CONFIGURATION Config0
  VAR_GLOBAL
    F_Conf : BOOL := TRUE;  (* Флаг конфигурирования *)
    F_Res : BOOL := FALSE;  (* Флаг готовности результата *)
    STAT : TStat;  (* Состояние выполнения *)
    HDR : THead;  (* Заголовок модели *)
    STS : TSets;  (* Массивы настроек *)
    ITS : TItems;  (* Массивы элементов *)
    SFC : ARRAY[0..2] OF TItem := [0, 0, 0];  (* Массив поверхностей *)
    CFG : TConf;  (* Заголовок трансформатора *)
    RAD : ARRAY[0..15] OF TRad := [0, 0, 0, 0, 0, 0, 0, 0, 0, 0, 0, 0, 0, 0, 0, 0];  (* Массив радиаторов *)
    VRI : TVarI;  (* Заголовок входа (24 байт) *)
    PHI : ARRAY[0..2] OF TPhaseI := [0, 0, 0];  (* Вход по фазам (3x32 байт) *)
    VRO : TVarO;  (* Заголовок выхода (24 байт) *)
    PHO : ARRAY[0..2] OF TPhaseO := [0, 0, 0];  (* Выход по фазам (3x32 байт) *)
    RES : TRes;  (* Заголовок расчёта *)
    rTest : REAL := 0.0;  (* Для отладки *)
  END_VAR
  RESOURCE Res0 ON PLC
    VAR_GLOBAL RETAIN
      MW0 AT %MW0 : UINT := 16#0000;  (* DEF[0].ID: = Трансформатор = *)
      MW1 AT %MW1 : UINT := 16#8000;  (* DEF[0].CF: Флаги (СК|ось|форма) *)
      MW2 AT %MW2 : UINT := 0;  (* DEF[0].R0: Начальный радиус *)
      MW3 AT %MW3 : UINT := 0;  (* DEF[0].XYZ[0]: Координата X *)
      MW4 AT %MW4 : UINT := 0;  (* DEF[0].XYZ[1]: Координата Y *)
      MW5 AT %MW5 : UINT := 0;  (* DEF[0].XYZ[2]: Координата Z *)
      MW6 AT %MW6 : UINT := 3600;  (* DEF[0].LWH[0]: Длина L *)
      MW7 AT %MW7 : UINT := 1240;  (* DEF[0].LWH[1]: Ширина W *)
      MW8 AT %MW8 : UINT := 3150;  (* DEF[0].LWH[2]: Высота H *)
      MW9 AT %MW9 : UINT := 16#7000;  (* DEF[0].GMV: #Grd(4)|#Mat(4)|#Val(8) *)
      MW10 AT %MW10 : UINT := 16#1000;  (* DEF[1].ID: = КОЖУХ = *)
      MW11 AT %MW11 : UINT := 16#8000;  (* DEF[1].CF: Флаги (СК|ось|форма) *)
      MW12 AT %MW12 : UINT := 0;  (* DEF[1].R0: Начальный радиус *)
      MW13 AT %MW13 : UINT := 0;  (* DEF[1].XYZ[0]: Координата X *)
      MW14 AT %MW14 : UINT := 0;  (* DEF[1].XYZ[1]: Координата Y *)
      MW15 AT %MW15 : UINT := 0;  (* DEF[1].XYZ[2]: Координата Z *)
      MW16 AT %MW16 : UINT := 3600;  (* DEF[1].LWH[0]: Длина L *)
      MW17 AT %MW17 : UINT := 1240;  (* DEF[1].LWH[1]: Ширина W *)
      MW18 AT %MW18 : UINT := 3150;  (* DEF[1].LWH[2]: Высота H *)
      MW19 AT %MW19 : UINT := 16#8000;  (* DEF[1].GMV: #Grd(4)|#Mat(4)|#Val(8) *)
      MW20 AT %MW20 : UINT := 16#1100;  (* DEF[2].ID: - Крышка (центр) *)
      MW21 AT %MW21 : UINT := 16#0000;  (* DEF[2].CF: Флаги (СК|ось|форма) *)
      MW22 AT %MW22 : UINT := 0;  (* DEF[2].R0: Начальный радиус *)
      MW23 AT %MW23 : UINT := 620;  (* DEF[2].XYZ[0]: Координата X *)
      MW24 AT %MW24 : UINT := 0;  (* DEF[2].XYZ[1]: Координата Y *)
      MW25 AT %MW25 : UINT := 3140;  (* DEF[2].XYZ[2]: Координата Z *)
      MW26 AT %MW26 : UINT := 2360;  (* DEF[2].LWH[0]: Длина L *)
      MW27 AT %MW27 : UINT := 1240;  (* DEF[2].LWH[1]: Ширина W *)
      MW28 AT %MW28 : UINT := 10;  (* DEF[2].LWH[2]: Высота H *)
      MW29 AT %MW29 : UINT := 16#8200;  (* DEF[2].GMV: #Grd(4)|#Mat(4)|#Val(8) *)
      MW30 AT %MW30 : UINT := 16#1200;  (* DEF[3].ID: - Крышка (лев) *)
      MW31 AT %MW31 : UINT := 16#7400;  (* DEF[3].CF: Флаги (СК|ось|форма) *)
      MW32 AT %MW32 : UINT := 0;  (* DEF[3].R0: Начальный радиус *)
      MW33 AT %MW33 : UINT := 620;  (* DEF[3].XYZ[0]: Координата X *)
      MW34 AT %MW34 : UINT := 620;  (* DEF[3].XYZ[1]: Координата Y *)
      MW35 AT %MW35 : UINT := 3140;  (* DEF[3].XYZ[2]: Координата Z *)
      MW36 AT %MW36 : UINT := 620;  (* DEF[3].LWH[0]: Длина L *)
      MW37 AT %MW37 : UINT := 180;  (* DEF[3].LWH[1]: Ширина W *)
      MW38 AT %MW38 : UINT := 10;  (* DEF[3].LWH[2]: Высота H *)
      MW39 AT %MW39 : UINT := 16#3200;  (* DEF[3].GMV: #Grd(4)|#Mat(4)|#Val(8) *)
      MW40 AT %MW40 : UINT := 16#1300;  (* DEF[4].ID: - Крышка (прав) *)
      MW41 AT %MW41 : UINT := 16#7C00;  (* DEF[4].CF: Флаги (СК|ось|форма) *)
      MW42 AT %MW42 : UINT := 0;  (* DEF[4].R0: Начальный радиус *)
      MW43 AT %MW43 : UINT := 2980;  (* DEF[4].XYZ[0]: Координата X *)
      MW44 AT %MW44 : UINT := 620;  (* DEF[4].XYZ[1]: Координата Y *)
      MW45 AT %MW45 : UINT := 3140;  (* DEF[4].XYZ[2]: Координата Z *)
      MW46 AT %MW46 : UINT := 620;  (* DEF[4].LWH[0]: Длина L *)
      MW47 AT %MW47 : UINT := 180;  (* DEF[4].LWH[1]: Ширина W *)
      MW48 AT %MW48 : UINT := 10;  (* DEF[4].LWH[2]: Высота H *)
      MW49 AT %MW49 : UINT := 16#3200;  (* DEF[4].GMV: #Grd(4)|#Mat(4)|#Val(8) *)
      MW50 AT %MW50 : UINT := 16#1400;  (* DEF[5].ID: - Днище (центр) *)
      MW51 AT %MW51 : UINT := 16#0000;  (* DEF[5].CF: Флаги (СК|ось|форма) *)
      MW52 AT %MW52 : UINT := 0;  (* DEF[5].R0: Начальный радиус *)
      MW53 AT %MW53 : UINT := 620;  (* DEF[5].XYZ[0]: Координата X *)
      MW54 AT %MW54 : UINT := 0;  (* DEF[5].XYZ[1]: Координата Y *)
      MW55 AT %MW55 : UINT := 0;  (* DEF[5].XYZ[2]: Координата Z *)
      MW56 AT %MW56 : UINT := 2360;  (* DEF[5].LWH[0]: Длина L *)
      MW57 AT %MW57 : UINT := 1240;  (* DEF[5].LWH[1]: Ширина W *)
      MW58 AT %MW58 : UINT := 10;  (* DEF[5].LWH[2]: Высота H *)
      MW59 AT %MW59 : UINT := 16#8200;  (* DEF[5].GMV: #Grd(4)|#Mat(4)|#Val(8) *)
      MW60 AT %MW60 : UINT := 16#1500;  (* DEF[6].ID: - Днище (лев) *)
      MW61 AT %MW61 : UINT := 16#7400;  (* DEF[6].CF: Флаги (СК|ось|форма) *)
      MW62 AT %MW62 : UINT := 0;  (* DEF[6].R0: Начальный радиус *)
      MW63 AT %MW63 : UINT := 620;  (* DEF[6].XYZ[0]: Координата X *)
      MW64 AT %MW64 : UINT := 620;  (* DEF[6].XYZ[1]: Координата Y *)
      MW65 AT %MW65 : UINT := 0;  (* DEF[6].XYZ[2]: Координата Z *)
      MW66 AT %MW66 : UINT := 620;  (* DEF[6].LWH[0]: Длина L *)
      MW67 AT %MW67 : UINT := 180;  (* DEF[6].LWH[1]: Ширина W *)
      MW68 AT %MW68 : UINT := 10;  (* DEF[6].LWH[2]: Высота H *)
      MW69 AT %MW69 : UINT := 16#3200;  (* DEF[6].GMV: #Grd(4)|#Mat(4)|#Val(8) *)
      MW70 AT %MW70 : UINT := 16#1600;  (* DEF[7].ID: - Днище (прав) *)
      MW71 AT %MW71 : UINT := 16#7C00;  (* DEF[7].CF: Флаги (СК|ось|форма) *)
      MW72 AT %MW72 : UINT := 0;  (* DEF[7].R0: Начальный радиус *)
      MW73 AT %MW73 : UINT := 2980;  (* DEF[7].XYZ[0]: Координата X *)
      MW74 AT %MW74 : UINT := 620;  (* DEF[7].XYZ[1]: Координата Y *)
      MW75 AT %MW75 : UINT := 0;  (* DEF[7].XYZ[2]: Координата Z *)
      MW76 AT %MW76 : UINT := 620;  (* DEF[7].LWH[0]: Длина L *)
      MW77 AT %MW77 : UINT := 180;  (* DEF[7].LWH[1]: Ширина W *)
      MW78 AT %MW78 : UINT := 10;  (* DEF[7].LWH[2]: Высота H *)
      MW79 AT %MW79 : UINT := 16#3200;  (* DEF[7].GMV: #Grd(4)|#Mat(4)|#Val(8) *)
      MW80 AT %MW80 : UINT := 16#1700;  (* DEF[8].ID: - Стенка левая *)
      MW81 AT %MW81 : UINT := 16#7400;  (* DEF[8].CF: Флаги (СК|ось|форма) *)
      MW82 AT %MW82 : UINT := 610;  (* DEF[8].R0: Начальный радиус *)
      MW83 AT %MW83 : UINT := 620;  (* DEF[8].XYZ[0]: Координата X *)
      MW84 AT %MW84 : UINT := 620;  (* DEF[8].XYZ[1]: Координата Y *)
      MW85 AT %MW85 : UINT := 10;  (* DEF[8].XYZ[2]: Координата Z *)
      MW86 AT %MW86 : UINT := 10;  (* DEF[8].LWH[0]: Длина L *)
      MW87 AT %MW87 : UINT := 180;  (* DEF[8].LWH[1]: Ширина W *)
      MW88 AT %MW88 : UINT := 3130;  (* DEF[8].LWH[2]: Высота H *)
      MW89 AT %MW89 : UINT := 16#1200;  (* DEF[8].GMV: #Grd(4)|#Mat(4)|#Val(8) *)
      MW90 AT %MW90 : UINT := 16#1800;  (* DEF[9].ID: - Стенка правая *)
      MW91 AT %MW91 : UINT := 16#7C00;  (* DEF[9].CF: Флаги (СК|ось|форма) *)
      MW92 AT %MW92 : UINT := 610;  (* DEF[9].R0: Начальный радиус *)
      MW93 AT %MW93 : UINT := 2980;  (* DEF[9].XYZ[0]: Координата X *)
      MW94 AT %MW94 : UINT := 620;  (* DEF[9].XYZ[1]: Координата Y *)
      MW95 AT %MW95 : UINT := 10;  (* DEF[9].XYZ[2]: Координата Z *)
      MW96 AT %MW96 : UINT := 10;  (* DEF[9].LWH[0]: Длина L *)
      MW97 AT %MW97 : UINT := 180;  (* DEF[9].LWH[1]: Ширина W *)
      MW98 AT %MW98 : UINT := 3130;  (* DEF[9].LWH[2]: Высота H *)
      MW99 AT %MW99 : UINT := 16#1200;  (* DEF[9].GMV: #Grd(4)|#Mat(4)|#Val(8) *)
      MW100 AT %MW100 : UINT := 16#1900;  (* DEF[10].ID: - Стенка передняя *)
      MW101 AT %MW101 : UINT := 16#0000;  (* DEF[10].CF: Флаги (СК|ось|форма) *)
      MW102 AT %MW102 : UINT := 0;  (* DEF[10].R0: Начальный радиус *)
      MW103 AT %MW103 : UINT := 620;  (* DEF[10].XYZ[0]: Координата X *)
      MW104 AT %MW104 : UINT := 0;  (* DEF[10].XYZ[1]: Координата Y *)
      MW105 AT %MW105 : UINT := 10;  (* DEF[10].XYZ[2]: Координата Z *)
      MW106 AT %MW106 : UINT := 2360;  (* DEF[10].LWH[0]: Длина L *)
      MW107 AT %MW107 : UINT := 10;  (* DEF[10].LWH[1]: Ширина W *)
      MW108 AT %MW108 : UINT := 3130;  (* DEF[10].LWH[2]: Высота H *)
      MW109 AT %MW109 : UINT := 16#7200;  (* DEF[10].GMV: #Grd(4)|#Mat(4)|#Val(8) *)
      MW110 AT %MW110 : UINT := 16#1A00;  (* DEF[11].ID: - Стенка задняя *)
      MW111 AT %MW111 : UINT := 16#0000;  (* DEF[11].CF: Флаги (СК|ось|форма) *)
      MW112 AT %MW112 : UINT := 0;  (* DEF[11].R0: Начальный радиус *)
      MW113 AT %MW113 : UINT := 620;  (* DEF[11].XYZ[0]: Координата X *)
      MW114 AT %MW114 : UINT := 1230;  (* DEF[11].XYZ[1]: Координата Y *)
      MW115 AT %MW115 : UINT := 10;  (* DEF[11].XYZ[2]: Координата Z *)
      MW116 AT %MW116 : UINT := 2360;  (* DEF[11].LWH[0]: Длина L *)
      MW117 AT %MW117 : UINT := 10;  (* DEF[11].LWH[1]: Ширина W *)
      MW118 AT %MW118 : UINT := 3130;  (* DEF[11].LWH[2]: Высота H *)
      MW119 AT %MW119 : UINT := 16#7200;  (* DEF[11].GMV: #Grd(4)|#Mat(4)|#Val(8) *)
      MW120 AT %MW120 : UINT := 16#1B00;  (* DEF[12].ID: - Масло слева *)
      MW121 AT %MW121 : UINT := 16#7400;  (* DEF[12].CF: Флаги (СК|ось|форма) *)
      MW122 AT %MW122 : UINT := 590;  (* DEF[12].R0: Начальный радиус *)
      MW123 AT %MW123 : UINT := 620;  (* DEF[12].XYZ[0]: Координата X *)
      MW124 AT %MW124 : UINT := 620;  (* DEF[12].XYZ[1]: Координата Y *)
      MW125 AT %MW125 : UINT := 10;  (* DEF[12].XYZ[2]: Координата Z *)
      MW126 AT %MW126 : UINT := 20;  (* DEF[12].LWH[0]: Длина L *)
      MW127 AT %MW127 : UINT := 180;  (* DEF[12].LWH[1]: Ширина W *)
      MW128 AT %MW128 : UINT := 3130;  (* DEF[12].LWH[2]: Высота H *)
      MW129 AT %MW129 : UINT := 16#1100;  (* DEF[12].GMV: #Grd(4)|#Mat(4)|#Val(8) *)
      MW130 AT %MW130 : UINT := 16#1C00;  (* DEF[13].ID: - Масло справа *)
      MW131 AT %MW131 : UINT := 16#7C00;  (* DEF[13].CF: Флаги (СК|ось|форма) *)
      MW132 AT %MW132 : UINT := 590;  (* DEF[13].R0: Начальный радиус *)
      MW133 AT %MW133 : UINT := 2980;  (* DEF[13].XYZ[0]: Координата X *)
      MW134 AT %MW134 : UINT := 620;  (* DEF[13].XYZ[1]: Координата Y *)
      MW135 AT %MW135 : UINT := 10;  (* DEF[13].XYZ[2]: Координата Z *)
      MW136 AT %MW136 : UINT := 20;  (* DEF[13].LWH[0]: Длина L *)
      MW137 AT %MW137 : UINT := 180;  (* DEF[13].LWH[1]: Ширина W *)
      MW138 AT %MW138 : UINT := 3130;  (* DEF[13].LWH[2]: Высота H *)
      MW139 AT %MW139 : UINT := 16#1100;  (* DEF[13].GMV: #Grd(4)|#Mat(4)|#Val(8) *)
      MW140 AT %MW140 : UINT := 16#1D00;  (* DEF[14].ID: - Масло спереди *)
      MW141 AT %MW141 : UINT := 16#0000;  (* DEF[14].CF: Флаги (СК|ось|форма) *)
      MW142 AT %MW142 : UINT := 0;  (* DEF[14].R0: Начальный радиус *)
      MW143 AT %MW143 : UINT := 620;  (* DEF[14].XYZ[0]: Координата X *)
      MW144 AT %MW144 : UINT := 10;  (* DEF[14].XYZ[1]: Координата Y *)
      MW145 AT %MW145 : UINT := 10;  (* DEF[14].XYZ[2]: Координата Z *)
      MW146 AT %MW146 : UINT := 2360;  (* DEF[14].LWH[0]: Длина L *)
      MW147 AT %MW147 : UINT := 20;  (* DEF[14].LWH[1]: Ширина W *)
      MW148 AT %MW148 : UINT := 3130;  (* DEF[14].LWH[2]: Высота H *)
      MW149 AT %MW149 : UINT := 16#7100;  (* DEF[14].GMV: #Grd(4)|#Mat(4)|#Val(8) *)
      MW150 AT %MW150 : UINT := 16#1E00;  (* DEF[15].ID: - Масло сзади *)
      MW151 AT %MW151 : UINT := 16#0000;  (* DEF[15].CF: Флаги (СК|ось|форма) *)
      MW152 AT %MW152 : UINT := 0;  (* DEF[15].R0: Начальный радиус *)
      MW153 AT %MW153 : UINT := 620;  (* DEF[15].XYZ[0]: Координата X *)
      MW154 AT %MW154 : UINT := 1210;  (* DEF[15].XYZ[1]: Координата Y *)
      MW155 AT %MW155 : UINT := 10;  (* DEF[15].XYZ[2]: Координата Z *)
      MW156 AT %MW156 : UINT := 2360;  (* DEF[15].LWH[0]: Длина L *)
      MW157 AT %MW157 : UINT := 20;  (* DEF[15].LWH[1]: Ширина W *)
      MW158 AT %MW158 : UINT := 3130;  (* DEF[15].LWH[2]: Высота H *)
      MW159 AT %MW159 : UINT := 16#7100;  (* DEF[15].GMV: #Grd(4)|#Mat(4)|#Val(8) *)
      MW160 AT %MW160 : UINT := 16#2000;  (* DEF[16].ID: = ЧЕРДАК = *)
      MW161 AT %MW161 : UINT := 16#8000;  (* DEF[16].CF: Флаги (СК|ось|форма) *)
      MW162 AT %MW162 : UINT := 0;  (* DEF[16].R0: Начальный радиус *)
      MW163 AT %MW163 : UINT := 30;  (* DEF[16].XYZ[0]: Координата X *)
      MW164 AT %MW164 : UINT := 30;  (* DEF[16].XYZ[1]: Координата Y *)
      MW165 AT %MW165 : UINT := 2400;  (* DEF[16].XYZ[2]: Координата Z *)
      MW166 AT %MW166 : UINT := 3540;  (* DEF[16].LWH[0]: Длина L *)
      MW167 AT %MW167 : UINT := 1180;  (* DEF[16].LWH[1]: Ширина W *)
      MW168 AT %MW168 : UINT := 740;  (* DEF[16].LWH[2]: Высота H *)
      MW169 AT %MW169 : UINT := 16#8000;  (* DEF[16].GMV: #Grd(4)|#Mat(4)|#Val(8) *)
      MW170 AT %MW170 : UINT := 16#2100;  (* DEF[17].ID: - Масло верх (центр) *)
      MW171 AT %MW171 : UINT := 16#0000;  (* DEF[17].CF: Флаги (СК|ось|форма) *)
      MW172 AT %MW172 : UINT := 0;  (* DEF[17].R0: Начальный радиус *)
      MW173 AT %MW173 : UINT := 590;  (* DEF[17].XYZ[0]: Координата X *)
      MW174 AT %MW174 : UINT := 0;  (* DEF[17].XYZ[1]: Координата Y *)
      MW175 AT %MW175 : UINT := 350;  (* DEF[17].XYZ[2]: Координата Z *)
      MW176 AT %MW176 : UINT := 2360;  (* DEF[17].LWH[0]: Длина L *)
      MW177 AT %MW177 : UINT := 1180;  (* DEF[17].LWH[1]: Ширина W *)
      MW178 AT %MW178 : UINT := 390;  (* DEF[17].LWH[2]: Высота H *)
      MW179 AT %MW179 : UINT := 16#8100;  (* DEF[17].GMV: #Grd(4)|#Mat(4)|#Val(8) *)
      MW180 AT %MW180 : UINT := 16#2200;  (* DEF[18].ID: - Масло верх (лев) *)
      MW181 AT %MW181 : UINT := 16#7400;  (* DEF[18].CF: Флаги (СК|ось|форма) *)
      MW182 AT %MW182 : UINT := 0;  (* DEF[18].R0: Начальный радиус *)
      MW183 AT %MW183 : UINT := 590;  (* DEF[18].XYZ[0]: Координата X *)
      MW184 AT %MW184 : UINT := 590;  (* DEF[18].XYZ[1]: Координата Y *)
      MW185 AT %MW185 : UINT := 350;  (* DEF[18].XYZ[2]: Координата Z *)
      MW186 AT %MW186 : UINT := 590;  (* DEF[18].LWH[0]: Длина L *)
      MW187 AT %MW187 : UINT := 180;  (* DEF[18].LWH[1]: Ширина W *)
      MW188 AT %MW188 : UINT := 390;  (* DEF[18].LWH[2]: Высота H *)
      MW189 AT %MW189 : UINT := 16#3100;  (* DEF[18].GMV: #Grd(4)|#Mat(4)|#Val(8) *)
      MW190 AT %MW190 : UINT := 16#2300;  (* DEF[19].ID: - Масло верх (прав) *)
      MW191 AT %MW191 : UINT := 16#7C00;  (* DEF[19].CF: Флаги (СК|ось|форма) *)
      MW192 AT %MW192 : UINT := 0;  (* DEF[19].R0: Начальный радиус *)
      MW193 AT %MW193 : UINT := 2950;  (* DEF[19].XYZ[0]: Координата X *)
      MW194 AT %MW194 : UINT := 590;  (* DEF[19].XYZ[1]: Координата Y *)
      MW195 AT %MW195 : UINT := 350;  (* DEF[19].XYZ[2]: Координата Z *)
      MW196 AT %MW196 : UINT := 590;  (* DEF[19].LWH[0]: Длина L *)
      MW197 AT %MW197 : UINT := 180;  (* DEF[19].LWH[1]: Ширина W *)
      MW198 AT %MW198 : UINT := 390;  (* DEF[19].LWH[2]: Высота H *)
      MW199 AT %MW199 : UINT := 16#3100;  (* DEF[19].GMV: #Grd(4)|#Mat(4)|#Val(8) *)
      MW200 AT %MW200 : UINT := 16#2400;  (* DEF[20].ID: = Ярмовой слой (верх) = *)
      MW201 AT %MW201 : UINT := 16#8000;  (* DEF[20].CF: Флаги (СК|ось|форма) *)
      MW202 AT %MW202 : UINT := 0;  (* DEF[20].R0: Начальный радиус *)
      MW203 AT %MW203 : UINT := 0;  (* DEF[20].XYZ[0]: Координата X *)
      MW204 AT %MW204 : UINT := 0;  (* DEF[20].XYZ[1]: Координата Y *)
      MW205 AT %MW205 : UINT := 0;  (* DEF[20].XYZ[2]: Координата Z *)
      MW206 AT %MW206 : UINT := 3540;  (* DEF[20].LWH[0]: Длина L *)
      MW207 AT %MW207 : UINT := 1180;  (* DEF[20].LWH[1]: Ширина W *)
      MW208 AT %MW208 : UINT := 350;  (* DEF[20].LWH[2]: Высота H *)
      MW209 AT %MW209 : UINT := 16#8000;  (* DEF[20].GMV: #Grd(4)|#Mat(4)|#Val(8) *)
      MW210 AT %MW210 : UINT := 16#2410;  (* DEF[21].ID: - Ярмо (верх) *)
      MW211 AT %MW211 : UINT := 16#0000;  (* DEF[21].CF: Флаги (СК|ось|форма) *)
      MW212 AT %MW212 : UINT := 0;  (* DEF[21].R0: Начальный радиус *)
      MW213 AT %MW213 : UINT := 275;  (* DEF[21].XYZ[0]: Координата X *)
      MW214 AT %MW214 : UINT := 275;  (* DEF[21].XYZ[1]: Координата Y *)
      MW215 AT %MW215 : UINT := 0;  (* DEF[21].XYZ[2]: Координата Z *)
      MW216 AT %MW216 : UINT := 2990;  (* DEF[21].LWH[0]: Длина L *)
      MW217 AT %MW217 : UINT := 630;  (* DEF[21].LWH[1]: Ширина W *)
      MW218 AT %MW218 : UINT := 350;  (* DEF[21].LWH[2]: Высота H *)
      MW219 AT %MW219 : UINT := 16#8300;  (* DEF[21].GMV: #Grd(4)|#Mat(4)|#Val(8) *)
      MW220 AT %MW220 : UINT := 16#2420;  (* DEF[22].ID: - Масло слева (верх) *)
      MW221 AT %MW221 : UINT := 16#7460;  (* DEF[22].CF: Флаги (СК|ось|форма) *)
      MW222 AT %MW222 : UINT := 315;  (* DEF[22].R0: Начальный радиус *)
      MW223 AT %MW223 : UINT := 590;  (* DEF[22].XYZ[0]: Координата X *)
      MW224 AT %MW224 : UINT := 590;  (* DEF[22].XYZ[1]: Координата Y *)
      MW225 AT %MW225 : UINT := 0;  (* DEF[22].XYZ[2]: Координата Z *)
      MW226 AT %MW226 : UINT := 275;  (* DEF[22].LWH[0]: Длина L *)
      MW227 AT %MW227 : UINT := 180;  (* DEF[22].LWH[1]: Ширина W *)
      MW228 AT %MW228 : UINT := 350;  (* DEF[22].LWH[2]: Высота H *)
      MW229 AT %MW229 : UINT := 16#3100;  (* DEF[22].GMV: #Grd(4)|#Mat(4)|#Val(8) *)
      MW230 AT %MW230 : UINT := 16#2430;  (* DEF[23].ID: - Масло справа (верх) *)
      MW231 AT %MW231 : UINT := 16#7C90;  (* DEF[23].CF: Флаги (СК|ось|форма) *)
      MW232 AT %MW232 : UINT := 315;  (* DEF[23].R0: Начальный радиус *)
      MW233 AT %MW233 : UINT := 2950;  (* DEF[23].XYZ[0]: Координата X *)
      MW234 AT %MW234 : UINT := 590;  (* DEF[23].XYZ[1]: Координата Y *)
      MW235 AT %MW235 : UINT := 0;  (* DEF[23].XYZ[2]: Координата Z *)
      MW236 AT %MW236 : UINT := 275;  (* DEF[23].LWH[0]: Длина L *)
      MW237 AT %MW237 : UINT := 180;  (* DEF[23].LWH[1]: Ширина W *)
      MW238 AT %MW238 : UINT := 350;  (* DEF[23].LWH[2]: Высота H *)
      MW239 AT %MW239 : UINT := 16#3100;  (* DEF[23].GMV: #Grd(4)|#Mat(4)|#Val(8) *)
      MW240 AT %MW240 : UINT := 16#2440;  (* DEF[24].ID: - Масло спереди (верх) *)
      MW241 AT %MW241 : UINT := 16#0000;  (* DEF[24].CF: Флаги (СК|ось|форма) *)
      MW242 AT %MW242 : UINT := 0;  (* DEF[24].R0: Начальный радиус *)
      MW243 AT %MW243 : UINT := 590;  (* DEF[24].XYZ[0]: Координата X *)
      MW244 AT %MW244 : UINT := 0;  (* DEF[24].XYZ[1]: Координата Y *)
      MW245 AT %MW245 : UINT := 0;  (* DEF[24].XYZ[2]: Координата Z *)
      MW246 AT %MW246 : UINT := 2360;  (* DEF[24].LWH[0]: Длина L *)
      MW247 AT %MW247 : UINT := 275;  (* DEF[24].LWH[1]: Ширина W *)
      MW248 AT %MW248 : UINT := 350;  (* DEF[24].LWH[2]: Высота H *)
      MW249 AT %MW249 : UINT := 16#8100;  (* DEF[24].GMV: #Grd(4)|#Mat(4)|#Val(8) *)
      MW250 AT %MW250 : UINT := 16#2450;  (* DEF[25].ID: - Масло сзади (верх) *)
      MW251 AT %MW251 : UINT := 16#0000;  (* DEF[25].CF: Флаги (СК|ось|форма) *)
      MW252 AT %MW252 : UINT := 0;  (* DEF[25].R0: Начальный радиус *)
      MW253 AT %MW253 : UINT := 590;  (* DEF[25].XYZ[0]: Координата X *)
      MW254 AT %MW254 : UINT := 905;  (* DEF[25].XYZ[1]: Координата Y *)
      MW255 AT %MW255 : UINT := 0;  (* DEF[25].XYZ[2]: Координата Z *)
      MW256 AT %MW256 : UINT := 2360;  (* DEF[25].LWH[0]: Длина L *)
      MW257 AT %MW257 : UINT := 275;  (* DEF[25].LWH[1]: Ширина W *)
      MW258 AT %MW258 : UINT := 350;  (* DEF[25].LWH[2]: Высота H *)
      MW259 AT %MW259 : UINT := 16#8100;  (* DEF[25].GMV: #Grd(4)|#Mat(4)|#Val(8) *)
      MW260 AT %MW260 : UINT := 16#3000;  (* DEF[26].ID: = ЦОКОЛЬ = *)
      MW261 AT %MW261 : UINT := 16#8000;  (* DEF[26].CF: Флаги (СК|ось|форма) *)
      MW262 AT %MW262 : UINT := 0;  (* DEF[26].R0: Начальный радиус *)
      MW263 AT %MW263 : UINT := 30;  (* DEF[26].XYZ[0]: Координата X *)
      MW264 AT %MW264 : UINT := 30;  (* DEF[26].XYZ[1]: Координата Y *)
      MW265 AT %MW265 : UINT := 10;  (* DEF[26].XYZ[2]: Координата Z *)
      MW266 AT %MW266 : UINT := 3540;  (* DEF[26].LWH[0]: Длина L *)
      MW267 AT %MW267 : UINT := 1180;  (* DEF[26].LWH[1]: Ширина W *)
      MW268 AT %MW268 : UINT := 390;  (* DEF[26].LWH[2]: Высота H *)
      MW269 AT %MW269 : UINT := 16#8000;  (* DEF[26].GMV: #Grd(4)|#Mat(4)|#Val(8) *)
      MW270 AT %MW270 : UINT := 16#3100;  (* DEF[27].ID: - Масло низ (центр) *)
      MW271 AT %MW271 : UINT := 16#0000;  (* DEF[27].CF: Флаги (СК|ось|форма) *)
      MW272 AT %MW272 : UINT := 0;  (* DEF[27].R0: Начальный радиус *)
      MW273 AT %MW273 : UINT := 590;  (* DEF[27].XYZ[0]: Координата X *)
      MW274 AT %MW274 : UINT := 0;  (* DEF[27].XYZ[1]: Координата Y *)
      MW275 AT %MW275 : UINT := 0;  (* DEF[27].XYZ[2]: Координата Z *)
      MW276 AT %MW276 : UINT := 2360;  (* DEF[27].LWH[0]: Длина L *)
      MW277 AT %MW277 : UINT := 1180;  (* DEF[27].LWH[1]: Ширина W *)
      MW278 AT %MW278 : UINT := 40;  (* DEF[27].LWH[2]: Высота H *)
      MW279 AT %MW279 : UINT := 16#8100;  (* DEF[27].GMV: #Grd(4)|#Mat(4)|#Val(8) *)
      MW280 AT %MW280 : UINT := 16#3200;  (* DEF[28].ID: - Масло низ (лев) *)
      MW281 AT %MW281 : UINT := 16#7400;  (* DEF[28].CF: Флаги (СК|ось|форма) *)
      MW282 AT %MW282 : UINT := 0;  (* DEF[28].R0: Начальный радиус *)
      MW283 AT %MW283 : UINT := 590;  (* DEF[28].XYZ[0]: Координата X *)
      MW284 AT %MW284 : UINT := 590;  (* DEF[28].XYZ[1]: Координата Y *)
      MW285 AT %MW285 : UINT := 0;  (* DEF[28].XYZ[2]: Координата Z *)
      MW286 AT %MW286 : UINT := 590;  (* DEF[28].LWH[0]: Длина L *)
      MW287 AT %MW287 : UINT := 180;  (* DEF[28].LWH[1]: Ширина W *)
      MW288 AT %MW288 : UINT := 40;  (* DEF[28].LWH[2]: Высота H *)
      MW289 AT %MW289 : UINT := 16#3100;  (* DEF[28].GMV: #Grd(4)|#Mat(4)|#Val(8) *)
      MW290 AT %MW290 : UINT := 16#3300;  (* DEF[29].ID: - Масло низ (прав) *)
      MW291 AT %MW291 : UINT := 16#7C00;  (* DEF[29].CF: Флаги (СК|ось|форма) *)
      MW292 AT %MW292 : UINT := 0;  (* DEF[29].R0: Начальный радиус *)
      MW293 AT %MW293 : UINT := 2950;  (* DEF[29].XYZ[0]: Координата X *)
      MW294 AT %MW294 : UINT := 590;  (* DEF[29].XYZ[1]: Координата Y *)
      MW295 AT %MW295 : UINT := 0;  (* DEF[29].XYZ[2]: Координата Z *)
      MW296 AT %MW296 : UINT := 590;  (* DEF[29].LWH[0]: Длина L *)
      MW297 AT %MW297 : UINT := 180;  (* DEF[29].LWH[1]: Ширина W *)
      MW298 AT %MW298 : UINT := 40;  (* DEF[29].LWH[2]: Высота H *)
      MW299 AT %MW299 : UINT := 16#3100;  (* DEF[29].GMV: #Grd(4)|#Mat(4)|#Val(8) *)
      MW300 AT %MW300 : UINT := 16#3400;  (* DEF[30].ID: = Ярмовой слой (низ) = *)
      MW301 AT %MW301 : UINT := 16#8000;  (* DEF[30].CF: Флаги (СК|ось|форма) *)
      MW302 AT %MW302 : UINT := 0;  (* DEF[30].R0: Начальный радиус *)
      MW303 AT %MW303 : UINT := 0;  (* DEF[30].XYZ[0]: Координата X *)
      MW304 AT %MW304 : UINT := 0;  (* DEF[30].XYZ[1]: Координата Y *)
      MW305 AT %MW305 : UINT := 40;  (* DEF[30].XYZ[2]: Координата Z *)
      MW306 AT %MW306 : UINT := 3540;  (* DEF[30].LWH[0]: Длина L *)
      MW307 AT %MW307 : UINT := 1180;  (* DEF[30].LWH[1]: Ширина W *)
      MW308 AT %MW308 : UINT := 350;  (* DEF[30].LWH[2]: Высота H *)
      MW309 AT %MW309 : UINT := 16#8000;  (* DEF[30].GMV: #Grd(4)|#Mat(4)|#Val(8) *)
      MW310 AT %MW310 : UINT := 16#3410;  (* DEF[31].ID: - Ярмо (низ) *)
      MW311 AT %MW311 : UINT := 16#0000;  (* DEF[31].CF: Флаги (СК|ось|форма) *)
      MW312 AT %MW312 : UINT := 0;  (* DEF[31].R0: Начальный радиус *)
      MW313 AT %MW313 : UINT := 275;  (* DEF[31].XYZ[0]: Координата X *)
      MW314 AT %MW314 : UINT := 275;  (* DEF[31].XYZ[1]: Координата Y *)
      MW315 AT %MW315 : UINT := 0;  (* DEF[31].XYZ[2]: Координата Z *)
      MW316 AT %MW316 : UINT := 2990;  (* DEF[31].LWH[0]: Длина L *)
      MW317 AT %MW317 : UINT := 630;  (* DEF[31].LWH[1]: Ширина W *)
      MW318 AT %MW318 : UINT := 350;  (* DEF[31].LWH[2]: Высота H *)
      MW319 AT %MW319 : UINT := 16#8300;  (* DEF[31].GMV: #Grd(4)|#Mat(4)|#Val(8) *)
      MW320 AT %MW320 : UINT := 16#3420;  (* DEF[32].ID: - Масло слева (низ) *)
      MW321 AT %MW321 : UINT := 16#7460;  (* DEF[32].CF: Флаги (СК|ось|форма) *)
      MW322 AT %MW322 : UINT := 315;  (* DEF[32].R0: Начальный радиус *)
      MW323 AT %MW323 : UINT := 590;  (* DEF[32].XYZ[0]: Координата X *)
      MW324 AT %MW324 : UINT := 590;  (* DEF[32].XYZ[1]: Координата Y *)
      MW325 AT %MW325 : UINT := 0;  (* DEF[32].XYZ[2]: Координата Z *)
      MW326 AT %MW326 : UINT := 275;  (* DEF[32].LWH[0]: Длина L *)
      MW327 AT %MW327 : UINT := 180;  (* DEF[32].LWH[1]: Ширина W *)
      MW328 AT %MW328 : UINT := 350;  (* DEF[32].LWH[2]: Высота H *)
      MW329 AT %MW329 : UINT := 16#3100;  (* DEF[32].GMV: #Grd(4)|#Mat(4)|#Val(8) *)
      MW330 AT %MW330 : UINT := 16#3430;  (* DEF[33].ID: - Масло справа (низ) *)
      MW331 AT %MW331 : UINT := 16#7C90;  (* DEF[33].CF: Флаги (СК|ось|форма) *)
      MW332 AT %MW332 : UINT := 315;  (* DEF[33].R0: Начальный радиус *)
      MW333 AT %MW333 : UINT := 2950;  (* DEF[33].XYZ[0]: Координата X *)
      MW334 AT %MW334 : UINT := 590;  (* DEF[33].XYZ[1]: Координата Y *)
      MW335 AT %MW335 : UINT := 0;  (* DEF[33].XYZ[2]: Координата Z *)
      MW336 AT %MW336 : UINT := 275;  (* DEF[33].LWH[0]: Длина L *)
      MW337 AT %MW337 : UINT := 180;  (* DEF[33].LWH[1]: Ширина W *)
      MW338 AT %MW338 : UINT := 350;  (* DEF[33].LWH[2]: Высота H *)
      MW339 AT %MW339 : UINT := 16#3100;  (* DEF[33].GMV: #Grd(4)|#Mat(4)|#Val(8) *)
      MW340 AT %MW340 : UINT := 16#3440;  (* DEF[34].ID: - Масло спереди (низ) *)
      MW341 AT %MW341 : UINT := 16#0000;  (* DEF[34].CF: Флаги (СК|ось|форма) *)
      MW342 AT %MW342 : UINT := 0;  (* DEF[34].R0: Начальный радиус *)
      MW343 AT %MW343 : UINT := 590;  (* DEF[34].XYZ[0]: Координата X *)
      MW344 AT %MW344 : UINT := 0;  (* DEF[34].XYZ[1]: Координата Y *)
      MW345 AT %MW345 : UINT := 0;  (* DEF[34].XYZ[2]: Координата Z *)
      MW346 AT %MW346 : UINT := 2360;  (* DEF[34].LWH[0]: Длина L *)
      MW347 AT %MW347 : UINT := 275;  (* DEF[34].LWH[1]: Ширина W *)
      MW348 AT %MW348 : UINT := 350;  (* DEF[34].LWH[2]: Высота H *)
      MW349 AT %MW349 : UINT := 16#8100;  (* DEF[34].GMV: #Grd(4)|#Mat(4)|#Val(8) *)
      MW350 AT %MW350 : UINT := 16#3450;  (* DEF[35].ID: - Масло сзади (низ) *)
      MW351 AT %MW351 : UINT := 16#0000;  (* DEF[35].CF: Флаги (СК|ось|форма) *)
      MW352 AT %MW352 : UINT := 0;  (* DEF[35].R0: Начальный радиус *)
      MW353 AT %MW353 : UINT := 590;  (* DEF[35].XYZ[0]: Координата X *)
      MW354 AT %MW354 : UINT := 905;  (* DEF[35].XYZ[1]: Координата Y *)
      MW355 AT %MW355 : UINT := 0;  (* DEF[35].XYZ[2]: Координата Z *)
      MW356 AT %MW356 : UINT := 2360;  (* DEF[35].LWH[0]: Длина L *)
      MW357 AT %MW357 : UINT := 275;  (* DEF[35].LWH[1]: Ширина W *)
      MW358 AT %MW358 : UINT := 350;  (* DEF[35].LWH[2]: Высота H *)
      MW359 AT %MW359 : UINT := 16#8100;  (* DEF[35].GMV: #Grd(4)|#Mat(4)|#Val(8) *)
      MW360 AT %MW360 : UINT := 16#4000;  (* DEF[36].ID: = АКТИВНАЯ ЗОНА = *)
      MW361 AT %MW361 : UINT := 16#8000;  (* DEF[36].CF: Флаги (СК|ось|форма) *)
      MW362 AT %MW362 : UINT := 0;  (* DEF[36].R0: Начальный радиус *)
      MW363 AT %MW363 : UINT := 30;  (* DEF[36].XYZ[0]: Координата X *)
      MW364 AT %MW364 : UINT := 30;  (* DEF[36].XYZ[1]: Координата Y *)
      MW365 AT %MW365 : UINT := 400;  (* DEF[36].XYZ[2]: Координата Z *)
      MW366 AT %MW366 : UINT := 3540;  (* DEF[36].LWH[0]: Длина L *)
      MW367 AT %MW367 : UINT := 1180;  (* DEF[36].LWH[1]: Ширина W *)
      MW368 AT %MW368 : UINT := 2000;  (* DEF[36].LWH[2]: Высота H *)
      MW369 AT %MW369 : UINT := 16#8000;  (* DEF[36].GMV: #Grd(4)|#Mat(4)|#Val(8) *)
      MW370 AT %MW370 : UINT := 16#4100;  (* DEF[37].ID: = Фаза 1 (лев) = *)
      MW371 AT %MW371 : UINT := 16#F009;  (* DEF[37].CF: Флаги (СК|ось|форма) *)
      MW372 AT %MW372 : UINT := 0;  (* DEF[37].R0: Начальный радиус *)
      MW373 AT %MW373 : UINT := 590;  (* DEF[37].XYZ[0]: Координата X *)
      MW374 AT %MW374 : UINT := 590;  (* DEF[37].XYZ[1]: Координата Y *)
      MW375 AT %MW375 : UINT := 0;  (* DEF[37].XYZ[2]: Координата Z *)
      MW376 AT %MW376 : UINT := 590;  (* DEF[37].LWH[0]: Длина L *)
      MW377 AT %MW377 : UINT := 360;  (* DEF[37].LWH[1]: Ширина W *)
      MW378 AT %MW378 : UINT := 2000;  (* DEF[37].LWH[2]: Высота H *)
      MW379 AT %MW379 : UINT := 16#1000;  (* DEF[37].GMV: #Grd(4)|#Mat(4)|#Val(8) *)
      MW380 AT %MW380 : UINT := 16#4110;  (* DEF[38].ID: - Стержень *)
      MW381 AT %MW381 : UINT := 16#4000;  (* DEF[38].CF: Флаги (СК|ось|форма) *)
      MW382 AT %MW382 : UINT := 0;  (* DEF[38].R0: Начальный радиус *)
      MW383 AT %MW383 : UINT := 0;  (* DEF[38].XYZ[0]: Координата X *)
      MW384 AT %MW384 : UINT := 0;  (* DEF[38].XYZ[1]: Координата Y *)
      MW385 AT %MW385 : UINT := 0;  (* DEF[38].XYZ[2]: Координата Z *)
      MW386 AT %MW386 : UINT := 315;  (* DEF[38].LWH[0]: Длина L *)
      MW387 AT %MW387 : UINT := 360;  (* DEF[38].LWH[1]: Ширина W *)
      MW388 AT %MW388 : UINT := 2000;  (* DEF[38].LWH[2]: Высота H *)
      MW389 AT %MW389 : UINT := 16#1300;  (* DEF[38].GMV: #Grd(4)|#Mat(4)|#Val(8) *)
      MW390 AT %MW390 : UINT := 16#4120;  (* DEF[39].ID: - Масло сверху *)
      MW391 AT %MW391 : UINT := 16#4009;  (* DEF[39].CF: Флаги (СК|ось|форма) *)
      MW392 AT %MW392 : UINT := 0;  (* DEF[39].R0: Начальный радиус *)
      MW393 AT %MW393 : UINT := 315;  (* DEF[39].XYZ[0]: Координата X *)
      MW394 AT %MW394 : UINT := 0;  (* DEF[39].XYZ[1]: Координата Y *)
      MW395 AT %MW395 : UINT := 1850;  (* DEF[39].XYZ[2]: Координата Z *)
      MW396 AT %MW396 : UINT := 275;  (* DEF[39].LWH[0]: Длина L *)
      MW397 AT %MW397 : UINT := 360;  (* DEF[39].LWH[1]: Ширина W *)
      MW398 AT %MW398 : UINT := 150;  (* DEF[39].LWH[2]: Высота H *)
      MW399 AT %MW399 : UINT := 16#5100;  (* DEF[39].GMV: #Grd(4)|#Mat(4)|#Val(8) *)
      MW400 AT %MW400 : UINT := 16#4130;  (* DEF[40].ID: - Масло снизу *)
      MW401 AT %MW401 : UINT := 16#4009;  (* DEF[40].CF: Флаги (СК|ось|форма) *)
      MW402 AT %MW402 : UINT := 0;  (* DEF[40].R0: Начальный радиус *)
      MW403 AT %MW403 : UINT := 315;  (* DEF[40].XYZ[0]: Координата X *)
      MW404 AT %MW404 : UINT := 0;  (* DEF[40].XYZ[1]: Координата Y *)
      MW405 AT %MW405 : UINT := 0;  (* DEF[40].XYZ[2]: Координата Z *)
      MW406 AT %MW406 : UINT := 275;  (* DEF[40].LWH[0]: Длина L *)
      MW407 AT %MW407 : UINT := 360;  (* DEF[40].LWH[1]: Ширина W *)
      MW408 AT %MW408 : UINT := 150;  (* DEF[40].LWH[2]: Высота H *)
      MW409 AT %MW409 : UINT := 16#5100;  (* DEF[40].GMV: #Grd(4)|#Mat(4)|#Val(8) *)
      MW410 AT %MW410 : UINT := 16#4140;  (* DEF[41].ID: - Маслоканал-1 *)
      MW411 AT %MW411 : UINT := 16#4000;  (* DEF[41].CF: Флаги (СК|ось|форма) *)
      MW412 AT %MW412 : UINT := 0;  (* DEF[41].R0: Начальный радиус *)
      MW413 AT %MW413 : UINT := 315;  (* DEF[41].XYZ[0]: Координата X *)
      MW414 AT %MW414 : UINT := 0;  (* DEF[41].XYZ[1]: Координата Y *)
      MW415 AT %MW415 : UINT := 150;  (* DEF[41].XYZ[2]: Координата Z *)
      MW416 AT %MW416 : UINT := 30;  (* DEF[41].LWH[0]: Длина L *)
      MW417 AT %MW417 : UINT := 360;  (* DEF[41].LWH[1]: Ширина W *)
      MW418 AT %MW418 : UINT := 1700;  (* DEF[41].LWH[2]: Высота H *)
      MW419 AT %MW419 : UINT := 16#1100;  (* DEF[41].GMV: #Grd(4)|#Mat(4)|#Val(8) *)
      MW420 AT %MW420 : UINT := 16#4150;  (* DEF[42].ID: - Обмотка НН *)
      MW421 AT %MW421 : UINT := 16#4000;  (* DEF[42].CF: Флаги (СК|ось|форма) *)
      MW422 AT %MW422 : UINT := 0;  (* DEF[42].R0: Начальный радиус *)
      MW423 AT %MW423 : UINT := 345;  (* DEF[42].XYZ[0]: Координата X *)
      MW424 AT %MW424 : UINT := 0;  (* DEF[42].XYZ[1]: Координата Y *)
      MW425 AT %MW425 : UINT := 150;  (* DEF[42].XYZ[2]: Координата Z *)
      MW426 AT %MW426 : UINT := 80;  (* DEF[42].LWH[0]: Длина L *)
      MW427 AT %MW427 : UINT := 360;  (* DEF[42].LWH[1]: Ширина W *)
      MW428 AT %MW428 : UINT := 1700;  (* DEF[42].LWH[2]: Высота H *)
      MW429 AT %MW429 : UINT := 16#1400;  (* DEF[42].GMV: #Grd(4)|#Mat(4)|#Val(8) *)
      MW430 AT %MW430 : UINT := 16#4160;  (* DEF[43].ID: - Маслоканал-2 *)
      MW431 AT %MW431 : UINT := 16#4000;  (* DEF[43].CF: Флаги (СК|ось|форма) *)
      MW432 AT %MW432 : UINT := 0;  (* DEF[43].R0: Начальный радиус *)
      MW433 AT %MW433 : UINT := 425;  (* DEF[43].XYZ[0]: Координата X *)
      MW434 AT %MW434 : UINT := 0;  (* DEF[43].XYZ[1]: Координата Y *)
      MW435 AT %MW435 : UINT := 150;  (* DEF[43].XYZ[2]: Координата Z *)
      MW436 AT %MW436 : UINT := 30;  (* DEF[43].LWH[0]: Длина L *)
      MW437 AT %MW437 : UINT := 360;  (* DEF[43].LWH[1]: Ширина W *)
      MW438 AT %MW438 : UINT := 1700;  (* DEF[43].LWH[2]: Высота H *)
      MW439 AT %MW439 : UINT := 16#1100;  (* DEF[43].GMV: #Grd(4)|#Mat(4)|#Val(8) *)
      MW440 AT %MW440 : UINT := 16#4170;  (* DEF[44].ID: = Обмотка ВН = *)
      MW441 AT %MW441 : UINT := 16#C000;  (* DEF[44].CF: Флаги (СК|ось|форма) *)
      MW442 AT %MW442 : UINT := 0;  (* DEF[44].R0: Начальный радиус *)
      MW443 AT %MW443 : UINT := 455;  (* DEF[44].XYZ[0]: Координата X *)
      MW444 AT %MW444 : UINT := 0;  (* DEF[44].XYZ[1]: Координата Y *)
      MW445 AT %MW445 : UINT := 150;  (* DEF[44].XYZ[2]: Координата Z *)
      MW446 AT %MW446 : UINT := 90;  (* DEF[44].LWH[0]: Длина L *)
      MW447 AT %MW447 : UINT := 360;  (* DEF[44].LWH[1]: Ширина W *)
      MW448 AT %MW448 : UINT := 1700;  (* DEF[44].LWH[2]: Высота H *)
      MW449 AT %MW449 : UINT := 16#1000;  (* DEF[44].GMV: #Grd(4)|#Mat(4)|#Val(8) *)
      MW450 AT %MW450 : UINT := 16#4171;  (* DEF[45].ID: - Катушка ВН-1 *)
      MW451 AT %MW451 : UINT := 16#4000;  (* DEF[45].CF: Флаги (СК|ось|форма) *)
      MW452 AT %MW452 : UINT := 0;  (* DEF[45].R0: Начальный радиус *)
      MW453 AT %MW453 : UINT := 455;  (* DEF[45].XYZ[0]: Координата X *)
      MW454 AT %MW454 : UINT := 0;  (* DEF[45].XYZ[1]: Координата Y *)
      MW455 AT %MW455 : UINT := 150;  (* DEF[45].XYZ[2]: Координата Z *)
      MW456 AT %MW456 : UINT := 90;  (* DEF[45].LWH[0]: Длина L *)
      MW457 AT %MW457 : UINT := 360;  (* DEF[45].LWH[1]: Ширина W *)
      MW458 AT %MW458 : UINT := 170;  (* DEF[45].LWH[2]: Высота H *)
      MW459 AT %MW459 : UINT := 16#3500;  (* DEF[45].GMV: #Grd(4)|#Mat(4)|#Val(8) *)
      MW460 AT %MW460 : UINT := 16#4172;  (* DEF[46].ID: - Катушка ВН-2 *)
      MW461 AT %MW461 : UINT := 16#4000;  (* DEF[46].CF: Флаги (СК|ось|форма) *)
      MW462 AT %MW462 : UINT := 0;  (* DEF[46].R0: Начальный радиус *)
      MW463 AT %MW463 : UINT := 455;  (* DEF[46].XYZ[0]: Координата X *)
      MW464 AT %MW464 : UINT := 0;  (* DEF[46].XYZ[1]: Координата Y *)
      MW465 AT %MW465 : UINT := 320;  (* DEF[46].XYZ[2]: Координата Z *)
      MW466 AT %MW466 : UINT := 90;  (* DEF[46].LWH[0]: Длина L *)
      MW467 AT %MW467 : UINT := 360;  (* DEF[46].LWH[1]: Ширина W *)
      MW468 AT %MW468 : UINT := 170;  (* DEF[46].LWH[2]: Высота H *)
      MW469 AT %MW469 : UINT := 16#3500;  (* DEF[46].GMV: #Grd(4)|#Mat(4)|#Val(8) *)
      MW470 AT %MW470 : UINT := 16#4173;  (* DEF[47].ID: - Катушка ВН-3 *)
      MW471 AT %MW471 : UINT := 16#4000;  (* DEF[47].CF: Флаги (СК|ось|форма) *)
      MW472 AT %MW472 : UINT := 0;  (* DEF[47].R0: Начальный радиус *)
      MW473 AT %MW473 : UINT := 455;  (* DEF[47].XYZ[0]: Координата X *)
      MW474 AT %MW474 : UINT := 0;  (* DEF[47].XYZ[1]: Координата Y *)
      MW475 AT %MW475 : UINT := 490;  (* DEF[47].XYZ[2]: Координата Z *)
      MW476 AT %MW476 : UINT := 90;  (* DEF[47].LWH[0]: Длина L *)
      MW477 AT %MW477 : UINT := 360;  (* DEF[47].LWH[1]: Ширина W *)
      MW478 AT %MW478 : UINT := 170;  (* DEF[47].LWH[2]: Высота H *)
      MW479 AT %MW479 : UINT := 16#3500;  (* DEF[47].GMV: #Grd(4)|#Mat(4)|#Val(8) *)
      MW480 AT %MW480 : UINT := 16#4174;  (* DEF[48].ID: - Катушка ВН-4 *)
      MW481 AT %MW481 : UINT := 16#4000;  (* DEF[48].CF: Флаги (СК|ось|форма) *)
      MW482 AT %MW482 : UINT := 0;  (* DEF[48].R0: Начальный радиус *)
      MW483 AT %MW483 : UINT := 455;  (* DEF[48].XYZ[0]: Координата X *)
      MW484 AT %MW484 : UINT := 0;  (* DEF[48].XYZ[1]: Координата Y *)
      MW485 AT %MW485 : UINT := 660;  (* DEF[48].XYZ[2]: Координата Z *)
      MW486 AT %MW486 : UINT := 90;  (* DEF[48].LWH[0]: Длина L *)
      MW487 AT %MW487 : UINT := 360;  (* DEF[48].LWH[1]: Ширина W *)
      MW488 AT %MW488 : UINT := 170;  (* DEF[48].LWH[2]: Высота H *)
      MW489 AT %MW489 : UINT := 16#3500;  (* DEF[48].GMV: #Grd(4)|#Mat(4)|#Val(8) *)
      MW490 AT %MW490 : UINT := 16#4175;  (* DEF[49].ID: - Катушка ВН-5 *)
      MW491 AT %MW491 : UINT := 16#4000;  (* DEF[49].CF: Флаги (СК|ось|форма) *)
      MW492 AT %MW492 : UINT := 0;  (* DEF[49].R0: Начальный радиус *)
      MW493 AT %MW493 : UINT := 455;  (* DEF[49].XYZ[0]: Координата X *)
      MW494 AT %MW494 : UINT := 0;  (* DEF[49].XYZ[1]: Координата Y *)
      MW495 AT %MW495 : UINT := 830;  (* DEF[49].XYZ[2]: Координата Z *)
      MW496 AT %MW496 : UINT := 90;  (* DEF[49].LWH[0]: Длина L *)
      MW497 AT %MW497 : UINT := 360;  (* DEF[49].LWH[1]: Ширина W *)
      MW498 AT %MW498 : UINT := 170;  (* DEF[49].LWH[2]: Высота H *)
      MW499 AT %MW499 : UINT := 16#3500;  (* DEF[49].GMV: #Grd(4)|#Mat(4)|#Val(8) *)
      MW500 AT %MW500 : UINT := 16#4176;  (* DEF[50].ID: - Катушка ВН-6 *)
      MW501 AT %MW501 : UINT := 16#4000;  (* DEF[50].CF: Флаги (СК|ось|форма) *)
      MW502 AT %MW502 : UINT := 0;  (* DEF[50].R0: Начальный радиус *)
      MW503 AT %MW503 : UINT := 455;  (* DEF[50].XYZ[0]: Координата X *)
      MW504 AT %MW504 : UINT := 0;  (* DEF[50].XYZ[1]: Координата Y *)
      MW505 AT %MW505 : UINT := 1000;  (* DEF[50].XYZ[2]: Координата Z *)
      MW506 AT %MW506 : UINT := 90;  (* DEF[50].LWH[0]: Длина L *)
      MW507 AT %MW507 : UINT := 360;  (* DEF[50].LWH[1]: Ширина W *)
      MW508 AT %MW508 : UINT := 170;  (* DEF[50].LWH[2]: Высота H *)
      MW509 AT %MW509 : UINT := 16#3500;  (* DEF[50].GMV: #Grd(4)|#Mat(4)|#Val(8) *)
      MW510 AT %MW510 : UINT := 16#4177;  (* DEF[51].ID: - Катушка ВН-7 *)
      MW511 AT %MW511 : UINT := 16#4000;  (* DEF[51].CF: Флаги (СК|ось|форма) *)
      MW512 AT %MW512 : UINT := 0;  (* DEF[51].R0: Начальный радиус *)
      MW513 AT %MW513 : UINT := 455;  (* DEF[51].XYZ[0]: Координата X *)
      MW514 AT %MW514 : UINT := 0;  (* DEF[51].XYZ[1]: Координата Y *)
      MW515 AT %MW515 : UINT := 1170;  (* DEF[51].XYZ[2]: Координата Z *)
      MW516 AT %MW516 : UINT := 90;  (* DEF[51].LWH[0]: Длина L *)
      MW517 AT %MW517 : UINT := 360;  (* DEF[51].LWH[1]: Ширина W *)
      MW518 AT %MW518 : UINT := 170;  (* DEF[51].LWH[2]: Высота H *)
      MW519 AT %MW519 : UINT := 16#3500;  (* DEF[51].GMV: #Grd(4)|#Mat(4)|#Val(8) *)
      MW520 AT %MW520 : UINT := 16#4178;  (* DEF[52].ID: - Катушка ВН-8 *)
      MW521 AT %MW521 : UINT := 16#4000;  (* DEF[52].CF: Флаги (СК|ось|форма) *)
      MW522 AT %MW522 : UINT := 0;  (* DEF[52].R0: Начальный радиус *)
      MW523 AT %MW523 : UINT := 455;  (* DEF[52].XYZ[0]: Координата X *)
      MW524 AT %MW524 : UINT := 0;  (* DEF[52].XYZ[1]: Координата Y *)
      MW525 AT %MW525 : UINT := 1340;  (* DEF[52].XYZ[2]: Координата Z *)
      MW526 AT %MW526 : UINT := 90;  (* DEF[52].LWH[0]: Длина L *)
      MW527 AT %MW527 : UINT := 360;  (* DEF[52].LWH[1]: Ширина W *)
      MW528 AT %MW528 : UINT := 170;  (* DEF[52].LWH[2]: Высота H *)
      MW529 AT %MW529 : UINT := 16#3500;  (* DEF[52].GMV: #Grd(4)|#Mat(4)|#Val(8) *)
      MW530 AT %MW530 : UINT := 16#4179;  (* DEF[53].ID: - Катушка ВН-9 *)
      MW531 AT %MW531 : UINT := 16#4000;  (* DEF[53].CF: Флаги (СК|ось|форма) *)
      MW532 AT %MW532 : UINT := 0;  (* DEF[53].R0: Начальный радиус *)
      MW533 AT %MW533 : UINT := 455;  (* DEF[53].XYZ[0]: Координата X *)
      MW534 AT %MW534 : UINT := 0;  (* DEF[53].XYZ[1]: Координата Y *)
      MW535 AT %MW535 : UINT := 1510;  (* DEF[53].XYZ[2]: Координата Z *)
      MW536 AT %MW536 : UINT := 90;  (* DEF[53].LWH[0]: Длина L *)
      MW537 AT %MW537 : UINT := 360;  (* DEF[53].LWH[1]: Ширина W *)
      MW538 AT %MW538 : UINT := 170;  (* DEF[53].LWH[2]: Высота H *)
      MW539 AT %MW539 : UINT := 16#3500;  (* DEF[53].GMV: #Grd(4)|#Mat(4)|#Val(8) *)
      MW540 AT %MW540 : UINT := 16#417A;  (* DEF[54].ID: - Катушка ВН-10 *)
      MW541 AT %MW541 : UINT := 16#4000;  (* DEF[54].CF: Флаги (СК|ось|форма) *)
      MW542 AT %MW542 : UINT := 0;  (* DEF[54].R0: Начальный радиус *)
      MW543 AT %MW543 : UINT := 455;  (* DEF[54].XYZ[0]: Координата X *)
      MW544 AT %MW544 : UINT := 0;  (* DEF[54].XYZ[1]: Координата Y *)
      MW545 AT %MW545 : UINT := 1680;  (* DEF[54].XYZ[2]: Координата Z *)
      MW546 AT %MW546 : UINT := 90;  (* DEF[54].LWH[0]: Длина L *)
      MW547 AT %MW547 : UINT := 360;  (* DEF[54].LWH[1]: Ширина W *)
      MW548 AT %MW548 : UINT := 170;  (* DEF[54].LWH[2]: Высота H *)
      MW549 AT %MW549 : UINT := 16#3500;  (* DEF[54].GMV: #Grd(4)|#Mat(4)|#Val(8) *)
      MW550 AT %MW550 : UINT := 16#4180;  (* DEF[55].ID: = Маслоканал-3 = *)
      MW551 AT %MW551 : UINT := 16#C009;  (* DEF[55].CF: Флаги (СК|ось|форма) *)
      MW552 AT %MW552 : UINT := 0;  (* DEF[55].R0: Начальный радиус *)
      MW553 AT %MW553 : UINT := 545;  (* DEF[55].XYZ[0]: Координата X *)
      MW554 AT %MW554 : UINT := 0;  (* DEF[55].XYZ[1]: Координата Y *)
      MW555 AT %MW555 : UINT := 150;  (* DEF[55].XYZ[2]: Координата Z *)
      MW556 AT %MW556 : UINT := 45;  (* DEF[55].LWH[0]: Длина L *)
      MW557 AT %MW557 : UINT := 360;  (* DEF[55].LWH[1]: Ширина W *)
      MW558 AT %MW558 : UINT := 1700;  (* DEF[55].LWH[2]: Высота H *)
      MW559 AT %MW559 : UINT := 16#1000;  (* DEF[55].GMV: #Grd(4)|#Mat(4)|#Val(8) *)
      MW560 AT %MW560 : UINT := 16#4181;  (* DEF[56].ID: - Маслоканал-3 (лев) *)
      MW561 AT %MW561 : UINT := 16#4000;  (* DEF[56].CF: Флаги (СК|ось|форма) *)
      MW562 AT %MW562 : UINT := 0;  (* DEF[56].R0: Начальный радиус *)
      MW563 AT %MW563 : UINT := 545;  (* DEF[56].XYZ[0]: Координата X *)
      MW564 AT %MW564 : UINT := 90;  (* DEF[56].XYZ[1]: Координата Y *)
      MW565 AT %MW565 : UINT := 150;  (* DEF[56].XYZ[2]: Координата Z *)
      MW566 AT %MW566 : UINT := 45;  (* DEF[56].LWH[0]: Длина L *)
      MW567 AT %MW567 : UINT := 180;  (* DEF[56].LWH[1]: Ширина W *)
      MW568 AT %MW568 : UINT := 1700;  (* DEF[56].LWH[2]: Высота H *)
      MW569 AT %MW569 : UINT := 16#1100;  (* DEF[56].GMV: #Grd(4)|#Mat(4)|#Val(8) *)
      MW570 AT %MW570 : UINT := 16#4182;  (* DEF[57].ID: - Маслоканал-3 (прав) *)
      MW571 AT %MW571 : UINT := 16#4009;  (* DEF[57].CF: Флаги (СК|ось|форма) *)
      MW572 AT %MW572 : UINT := 0;  (* DEF[57].R0: Начальный радиус *)
      MW573 AT %MW573 : UINT := 545;  (* DEF[57].XYZ[0]: Координата X *)
      MW574 AT %MW574 : UINT := -90;  (* DEF[57].XYZ[1]: Координата Y *)
      MW575 AT %MW575 : UINT := 150;  (* DEF[57].XYZ[2]: Координата Z *)
      MW576 AT %MW576 : UINT := 45;  (* DEF[57].LWH[0]: Длина L *)
      MW577 AT %MW577 : UINT := 180;  (* DEF[57].LWH[1]: Ширина W *)
      MW578 AT %MW578 : UINT := 1700;  (* DEF[57].LWH[2]: Высота H *)
      MW579 AT %MW579 : UINT := 16#1100;  (* DEF[57].GMV: #Grd(4)|#Mat(4)|#Val(8) *)
      MW580 AT %MW580 : UINT := 16#4200;  (* DEF[58].ID: = Фаза 2 (центр) *)
      MW581 AT %MW581 : UINT := 16#F00F;  (* DEF[58].CF: Флаги (СК|ось|форма) *)
      MW582 AT %MW582 : UINT := 0;  (* DEF[58].R0: Начальный радиус *)
      MW583 AT %MW583 : UINT := 1770;  (* DEF[58].XYZ[0]: Координата X *)
      MW584 AT %MW584 : UINT := 590;  (* DEF[58].XYZ[1]: Координата Y *)
      MW585 AT %MW585 : UINT := 0;  (* DEF[58].XYZ[2]: Координата Z *)
      MW586 AT %MW586 : UINT := 590;  (* DEF[58].LWH[0]: Длина L *)
      MW587 AT %MW587 : UINT := 360;  (* DEF[58].LWH[1]: Ширина W *)
      MW588 AT %MW588 : UINT := 2000;  (* DEF[58].LWH[2]: Высота H *)
      MW589 AT %MW589 : UINT := 16#1000;  (* DEF[58].GMV: #Grd(4)|#Mat(4)|#Val(8) *)
      MW590 AT %MW590 : UINT := 16#4210;  (* DEF[59].ID: - Стержень *)
      MW591 AT %MW591 : UINT := 16#4000;  (* DEF[59].CF: Флаги (СК|ось|форма) *)
      MW592 AT %MW592 : UINT := 0;  (* DEF[59].R0: Начальный радиус *)
      MW593 AT %MW593 : UINT := 0;  (* DEF[59].XYZ[0]: Координата X *)
      MW594 AT %MW594 : UINT := 0;  (* DEF[59].XYZ[1]: Координата Y *)
      MW595 AT %MW595 : UINT := 0;  (* DEF[59].XYZ[2]: Координата Z *)
      MW596 AT %MW596 : UINT := 315;  (* DEF[59].LWH[0]: Длина L *)
      MW597 AT %MW597 : UINT := 360;  (* DEF[59].LWH[1]: Ширина W *)
      MW598 AT %MW598 : UINT := 2000;  (* DEF[59].LWH[2]: Высота H *)
      MW599 AT %MW599 : UINT := 16#1300;  (* DEF[59].GMV: #Grd(4)|#Mat(4)|#Val(8) *)
      MW600 AT %MW600 : UINT := 16#4220;  (* DEF[60].ID: - Масло сверху *)
      MW601 AT %MW601 : UINT := 16#400F;  (* DEF[60].CF: Флаги (СК|ось|форма) *)
      MW602 AT %MW602 : UINT := 0;  (* DEF[60].R0: Начальный радиус *)
      MW603 AT %MW603 : UINT := 315;  (* DEF[60].XYZ[0]: Координата X *)
      MW604 AT %MW604 : UINT := 0;  (* DEF[60].XYZ[1]: Координата Y *)
      MW605 AT %MW605 : UINT := 1850;  (* DEF[60].XYZ[2]: Координата Z *)
      MW606 AT %MW606 : UINT := 275;  (* DEF[60].LWH[0]: Длина L *)
      MW607 AT %MW607 : UINT := 360;  (* DEF[60].LWH[1]: Ширина W *)
      MW608 AT %MW608 : UINT := 150;  (* DEF[60].LWH[2]: Высота H *)
      MW609 AT %MW609 : UINT := 16#5100;  (* DEF[60].GMV: #Grd(4)|#Mat(4)|#Val(8) *)
      MW610 AT %MW610 : UINT := 16#4230;  (* DEF[61].ID: - Масло снизу *)
      MW611 AT %MW611 : UINT := 16#400F;  (* DEF[61].CF: Флаги (СК|ось|форма) *)
      MW612 AT %MW612 : UINT := 0;  (* DEF[61].R0: Начальный радиус *)
      MW613 AT %MW613 : UINT := 315;  (* DEF[61].XYZ[0]: Координата X *)
      MW614 AT %MW614 : UINT := 0;  (* DEF[61].XYZ[1]: Координата Y *)
      MW615 AT %MW615 : UINT := 0;  (* DEF[61].XYZ[2]: Координата Z *)
      MW616 AT %MW616 : UINT := 275;  (* DEF[61].LWH[0]: Длина L *)
      MW617 AT %MW617 : UINT := 360;  (* DEF[61].LWH[1]: Ширина W *)
      MW618 AT %MW618 : UINT := 150;  (* DEF[61].LWH[2]: Высота H *)
      MW619 AT %MW619 : UINT := 16#5100;  (* DEF[61].GMV: #Grd(4)|#Mat(4)|#Val(8) *)
      MW620 AT %MW620 : UINT := 16#4240;  (* DEF[62].ID: - Маслоканал-1 *)
      MW621 AT %MW621 : UINT := 16#4000;  (* DEF[62].CF: Флаги (СК|ось|форма) *)
      MW622 AT %MW622 : UINT := 0;  (* DEF[62].R0: Начальный радиус *)
      MW623 AT %MW623 : UINT := 315;  (* DEF[62].XYZ[0]: Координата X *)
      MW624 AT %MW624 : UINT := 0;  (* DEF[62].XYZ[1]: Координата Y *)
      MW625 AT %MW625 : UINT := 150;  (* DEF[62].XYZ[2]: Координата Z *)
      MW626 AT %MW626 : UINT := 30;  (* DEF[62].LWH[0]: Длина L *)
      MW627 AT %MW627 : UINT := 360;  (* DEF[62].LWH[1]: Ширина W *)
      MW628 AT %MW628 : UINT := 1700;  (* DEF[62].LWH[2]: Высота H *)
      MW629 AT %MW629 : UINT := 16#1100;  (* DEF[62].GMV: #Grd(4)|#Mat(4)|#Val(8) *)
      MW630 AT %MW630 : UINT := 16#4250;  (* DEF[63].ID: - Обмотка НН *)
      MW631 AT %MW631 : UINT := 16#4000;  (* DEF[63].CF: Флаги (СК|ось|форма) *)
      MW632 AT %MW632 : UINT := 0;  (* DEF[63].R0: Начальный радиус *)
      MW633 AT %MW633 : UINT := 345;  (* DEF[63].XYZ[0]: Координата X *)
      MW634 AT %MW634 : UINT := 0;  (* DEF[63].XYZ[1]: Координата Y *)
      MW635 AT %MW635 : UINT := 150;  (* DEF[63].XYZ[2]: Координата Z *)
      MW636 AT %MW636 : UINT := 80;  (* DEF[63].LWH[0]: Длина L *)
      MW637 AT %MW637 : UINT := 360;  (* DEF[63].LWH[1]: Ширина W *)
      MW638 AT %MW638 : UINT := 1700;  (* DEF[63].LWH[2]: Высота H *)
      MW639 AT %MW639 : UINT := 16#1400;  (* DEF[63].GMV: #Grd(4)|#Mat(4)|#Val(8) *)
      MW640 AT %MW640 : UINT := 16#4260;  (* DEF[64].ID: - Маслоканал-2 *)
      MW641 AT %MW641 : UINT := 16#4000;  (* DEF[64].CF: Флаги (СК|ось|форма) *)
      MW642 AT %MW642 : UINT := 0;  (* DEF[64].R0: Начальный радиус *)
      MW643 AT %MW643 : UINT := 425;  (* DEF[64].XYZ[0]: Координата X *)
      MW644 AT %MW644 : UINT := 0;  (* DEF[64].XYZ[1]: Координата Y *)
      MW645 AT %MW645 : UINT := 150;  (* DEF[64].XYZ[2]: Координата Z *)
      MW646 AT %MW646 : UINT := 30;  (* DEF[64].LWH[0]: Длина L *)
      MW647 AT %MW647 : UINT := 360;  (* DEF[64].LWH[1]: Ширина W *)
      MW648 AT %MW648 : UINT := 1700;  (* DEF[64].LWH[2]: Высота H *)
      MW649 AT %MW649 : UINT := 16#1100;  (* DEF[64].GMV: #Grd(4)|#Mat(4)|#Val(8) *)
      MW650 AT %MW650 : UINT := 16#4270;  (* DEF[65].ID: = Обмотка ВН = *)
      MW651 AT %MW651 : UINT := 16#C000;  (* DEF[65].CF: Флаги (СК|ось|форма) *)
      MW652 AT %MW652 : UINT := 0;  (* DEF[65].R0: Начальный радиус *)
      MW653 AT %MW653 : UINT := 455;  (* DEF[65].XYZ[0]: Координата X *)
      MW654 AT %MW654 : UINT := 0;  (* DEF[65].XYZ[1]: Координата Y *)
      MW655 AT %MW655 : UINT := 150;  (* DEF[65].XYZ[2]: Координата Z *)
      MW656 AT %MW656 : UINT := 90;  (* DEF[65].LWH[0]: Длина L *)
      MW657 AT %MW657 : UINT := 360;  (* DEF[65].LWH[1]: Ширина W *)
      MW658 AT %MW658 : UINT := 1700;  (* DEF[65].LWH[2]: Высота H *)
      MW659 AT %MW659 : UINT := 16#1000;  (* DEF[65].GMV: #Grd(4)|#Mat(4)|#Val(8) *)
      MW660 AT %MW660 : UINT := 16#4271;  (* DEF[66].ID: - Катушка ВН-1 *)
      MW661 AT %MW661 : UINT := 16#4000;  (* DEF[66].CF: Флаги (СК|ось|форма) *)
      MW662 AT %MW662 : UINT := 0;  (* DEF[66].R0: Начальный радиус *)
      MW663 AT %MW663 : UINT := 455;  (* DEF[66].XYZ[0]: Координата X *)
      MW664 AT %MW664 : UINT := 0;  (* DEF[66].XYZ[1]: Координата Y *)
      MW665 AT %MW665 : UINT := 150;  (* DEF[66].XYZ[2]: Координата Z *)
      MW666 AT %MW666 : UINT := 90;  (* DEF[66].LWH[0]: Длина L *)
      MW667 AT %MW667 : UINT := 360;  (* DEF[66].LWH[1]: Ширина W *)
      MW668 AT %MW668 : UINT := 170;  (* DEF[66].LWH[2]: Высота H *)
      MW669 AT %MW669 : UINT := 16#3500;  (* DEF[66].GMV: #Grd(4)|#Mat(4)|#Val(8) *)
      MW670 AT %MW670 : UINT := 16#4272;  (* DEF[67].ID: - Катушка ВН-2 *)
      MW671 AT %MW671 : UINT := 16#4000;  (* DEF[67].CF: Флаги (СК|ось|форма) *)
      MW672 AT %MW672 : UINT := 0;  (* DEF[67].R0: Начальный радиус *)
      MW673 AT %MW673 : UINT := 455;  (* DEF[67].XYZ[0]: Координата X *)
      MW674 AT %MW674 : UINT := 0;  (* DEF[67].XYZ[1]: Координата Y *)
      MW675 AT %MW675 : UINT := 320;  (* DEF[67].XYZ[2]: Координата Z *)
      MW676 AT %MW676 : UINT := 90;  (* DEF[67].LWH[0]: Длина L *)
      MW677 AT %MW677 : UINT := 360;  (* DEF[67].LWH[1]: Ширина W *)
      MW678 AT %MW678 : UINT := 170;  (* DEF[67].LWH[2]: Высота H *)
      MW679 AT %MW679 : UINT := 16#3500;  (* DEF[67].GMV: #Grd(4)|#Mat(4)|#Val(8) *)
      MW680 AT %MW680 : UINT := 16#4273;  (* DEF[68].ID: - Катушка ВН-3 *)
      MW681 AT %MW681 : UINT := 16#4000;  (* DEF[68].CF: Флаги (СК|ось|форма) *)
      MW682 AT %MW682 : UINT := 0;  (* DEF[68].R0: Начальный радиус *)
      MW683 AT %MW683 : UINT := 455;  (* DEF[68].XYZ[0]: Координата X *)
      MW684 AT %MW684 : UINT := 0;  (* DEF[68].XYZ[1]: Координата Y *)
      MW685 AT %MW685 : UINT := 490;  (* DEF[68].XYZ[2]: Координата Z *)
      MW686 AT %MW686 : UINT := 90;  (* DEF[68].LWH[0]: Длина L *)
      MW687 AT %MW687 : UINT := 360;  (* DEF[68].LWH[1]: Ширина W *)
      MW688 AT %MW688 : UINT := 170;  (* DEF[68].LWH[2]: Высота H *)
      MW689 AT %MW689 : UINT := 16#3500;  (* DEF[68].GMV: #Grd(4)|#Mat(4)|#Val(8) *)
      MW690 AT %MW690 : UINT := 16#4274;  (* DEF[69].ID: - Катушка ВН-4 *)
      MW691 AT %MW691 : UINT := 16#4000;  (* DEF[69].CF: Флаги (СК|ось|форма) *)
      MW692 AT %MW692 : UINT := 0;  (* DEF[69].R0: Начальный радиус *)
      MW693 AT %MW693 : UINT := 455;  (* DEF[69].XYZ[0]: Координата X *)
      MW694 AT %MW694 : UINT := 0;  (* DEF[69].XYZ[1]: Координата Y *)
      MW695 AT %MW695 : UINT := 660;  (* DEF[69].XYZ[2]: Координата Z *)
      MW696 AT %MW696 : UINT := 90;  (* DEF[69].LWH[0]: Длина L *)
      MW697 AT %MW697 : UINT := 360;  (* DEF[69].LWH[1]: Ширина W *)
      MW698 AT %MW698 : UINT := 170;  (* DEF[69].LWH[2]: Высота H *)
      MW699 AT %MW699 : UINT := 16#3500;  (* DEF[69].GMV: #Grd(4)|#Mat(4)|#Val(8) *)
      MW700 AT %MW700 : UINT := 16#4275;  (* DEF[70].ID: - Катушка ВН-5 *)
      MW701 AT %MW701 : UINT := 16#4000;  (* DEF[70].CF: Флаги (СК|ось|форма) *)
      MW702 AT %MW702 : UINT := 0;  (* DEF[70].R0: Начальный радиус *)
      MW703 AT %MW703 : UINT := 455;  (* DEF[70].XYZ[0]: Координата X *)
      MW704 AT %MW704 : UINT := 0;  (* DEF[70].XYZ[1]: Координата Y *)
      MW705 AT %MW705 : UINT := 830;  (* DEF[70].XYZ[2]: Координата Z *)
      MW706 AT %MW706 : UINT := 90;  (* DEF[70].LWH[0]: Длина L *)
      MW707 AT %MW707 : UINT := 360;  (* DEF[70].LWH[1]: Ширина W *)
      MW708 AT %MW708 : UINT := 170;  (* DEF[70].LWH[2]: Высота H *)
      MW709 AT %MW709 : UINT := 16#3500;  (* DEF[70].GMV: #Grd(4)|#Mat(4)|#Val(8) *)
      MW710 AT %MW710 : UINT := 16#4276;  (* DEF[71].ID: - Катушка ВН-6 *)
      MW711 AT %MW711 : UINT := 16#4000;  (* DEF[71].CF: Флаги (СК|ось|форма) *)
      MW712 AT %MW712 : UINT := 0;  (* DEF[71].R0: Начальный радиус *)
      MW713 AT %MW713 : UINT := 455;  (* DEF[71].XYZ[0]: Координата X *)
      MW714 AT %MW714 : UINT := 0;  (* DEF[71].XYZ[1]: Координата Y *)
      MW715 AT %MW715 : UINT := 1000;  (* DEF[71].XYZ[2]: Координата Z *)
      MW716 AT %MW716 : UINT := 90;  (* DEF[71].LWH[0]: Длина L *)
      MW717 AT %MW717 : UINT := 360;  (* DEF[71].LWH[1]: Ширина W *)
      MW718 AT %MW718 : UINT := 170;  (* DEF[71].LWH[2]: Высота H *)
      MW719 AT %MW719 : UINT := 16#3500;  (* DEF[71].GMV: #Grd(4)|#Mat(4)|#Val(8) *)
      MW720 AT %MW720 : UINT := 16#4277;  (* DEF[72].ID: - Катушка ВН-7 *)
      MW721 AT %MW721 : UINT := 16#4000;  (* DEF[72].CF: Флаги (СК|ось|форма) *)
      MW722 AT %MW722 : UINT := 0;  (* DEF[72].R0: Начальный радиус *)
      MW723 AT %MW723 : UINT := 455;  (* DEF[72].XYZ[0]: Координата X *)
      MW724 AT %MW724 : UINT := 0;  (* DEF[72].XYZ[1]: Координата Y *)
      MW725 AT %MW725 : UINT := 1170;  (* DEF[72].XYZ[2]: Координата Z *)
      MW726 AT %MW726 : UINT := 90;  (* DEF[72].LWH[0]: Длина L *)
      MW727 AT %MW727 : UINT := 360;  (* DEF[72].LWH[1]: Ширина W *)
      MW728 AT %MW728 : UINT := 170;  (* DEF[72].LWH[2]: Высота H *)
      MW729 AT %MW729 : UINT := 16#3500;  (* DEF[72].GMV: #Grd(4)|#Mat(4)|#Val(8) *)
      MW730 AT %MW730 : UINT := 16#4278;  (* DEF[73].ID: - Катушка ВН-8 *)
      MW731 AT %MW731 : UINT := 16#4000;  (* DEF[73].CF: Флаги (СК|ось|форма) *)
      MW732 AT %MW732 : UINT := 0;  (* DEF[73].R0: Начальный радиус *)
      MW733 AT %MW733 : UINT := 455;  (* DEF[73].XYZ[0]: Координата X *)
      MW734 AT %MW734 : UINT := 0;  (* DEF[73].XYZ[1]: Координата Y *)
      MW735 AT %MW735 : UINT := 1340;  (* DEF[73].XYZ[2]: Координата Z *)
      MW736 AT %MW736 : UINT := 90;  (* DEF[73].LWH[0]: Длина L *)
      MW737 AT %MW737 : UINT := 360;  (* DEF[73].LWH[1]: Ширина W *)
      MW738 AT %MW738 : UINT := 170;  (* DEF[73].LWH[2]: Высота H *)
      MW739 AT %MW739 : UINT := 16#3500;  (* DEF[73].GMV: #Grd(4)|#Mat(4)|#Val(8) *)
      MW740 AT %MW740 : UINT := 16#4279;  (* DEF[74].ID: - Катушка ВН-9 *)
      MW741 AT %MW741 : UINT := 16#4000;  (* DEF[74].CF: Флаги (СК|ось|форма) *)
      MW742 AT %MW742 : UINT := 0;  (* DEF[74].R0: Начальный радиус *)
      MW743 AT %MW743 : UINT := 455;  (* DEF[74].XYZ[0]: Координата X *)
      MW744 AT %MW744 : UINT := 0;  (* DEF[74].XYZ[1]: Координата Y *)
      MW745 AT %MW745 : UINT := 1510;  (* DEF[74].XYZ[2]: Координата Z *)
      MW746 AT %MW746 : UINT := 90;  (* DEF[74].LWH[0]: Длина L *)
      MW747 AT %MW747 : UINT := 360;  (* DEF[74].LWH[1]: Ширина W *)
      MW748 AT %MW748 : UINT := 170;  (* DEF[74].LWH[2]: Высота H *)
      MW749 AT %MW749 : UINT := 16#3500;  (* DEF[74].GMV: #Grd(4)|#Mat(4)|#Val(8) *)
      MW750 AT %MW750 : UINT := 16#427A;  (* DEF[75].ID: - Катушка ВН-10 *)
      MW751 AT %MW751 : UINT := 16#4000;  (* DEF[75].CF: Флаги (СК|ось|форма) *)
      MW752 AT %MW752 : UINT := 0;  (* DEF[75].R0: Начальный радиус *)
      MW753 AT %MW753 : UINT := 455;  (* DEF[75].XYZ[0]: Координата X *)
      MW754 AT %MW754 : UINT := 0;  (* DEF[75].XYZ[1]: Координата Y *)
      MW755 AT %MW755 : UINT := 1680;  (* DEF[75].XYZ[2]: Координата Z *)
      MW756 AT %MW756 : UINT := 90;  (* DEF[75].LWH[0]: Длина L *)
      MW757 AT %MW757 : UINT := 360;  (* DEF[75].LWH[1]: Ширина W *)
      MW758 AT %MW758 : UINT := 170;  (* DEF[75].LWH[2]: Высота H *)
      MW759 AT %MW759 : UINT := 16#3500;  (* DEF[75].GMV: #Grd(4)|#Mat(4)|#Val(8) *)
      MW760 AT %MW760 : UINT := 16#4280;  (* DEF[76].ID: = Маслоканал-3 = *)
      MW761 AT %MW761 : UINT := 16#C00F;  (* DEF[76].CF: Флаги (СК|ось|форма) *)
      MW762 AT %MW762 : UINT := 0;  (* DEF[76].R0: Начальный радиус *)
      MW763 AT %MW763 : UINT := 545;  (* DEF[76].XYZ[0]: Координата X *)
      MW764 AT %MW764 : UINT := 0;  (* DEF[76].XYZ[1]: Координата Y *)
      MW765 AT %MW765 : UINT := 150;  (* DEF[76].XYZ[2]: Координата Z *)
      MW766 AT %MW766 : UINT := 45;  (* DEF[76].LWH[0]: Длина L *)
      MW767 AT %MW767 : UINT := 360;  (* DEF[76].LWH[1]: Ширина W *)
      MW768 AT %MW768 : UINT := 1700;  (* DEF[76].LWH[2]: Высота H *)
      MW769 AT %MW769 : UINT := 16#1000;  (* DEF[76].GMV: #Grd(4)|#Mat(4)|#Val(8) *)
      MW770 AT %MW770 : UINT := 16#4281;  (* DEF[77].ID: - Маслоканал-3 (лев) *)
      MW771 AT %MW771 : UINT := 16#400F;  (* DEF[77].CF: Флаги (СК|ось|форма) *)
      MW772 AT %MW772 : UINT := 0;  (* DEF[77].R0: Начальный радиус *)
      MW773 AT %MW773 : UINT := 545;  (* DEF[77].XYZ[0]: Координата X *)
      MW774 AT %MW774 : UINT := 90;  (* DEF[77].XYZ[1]: Координата Y *)
      MW775 AT %MW775 : UINT := 150;  (* DEF[77].XYZ[2]: Координата Z *)
      MW776 AT %MW776 : UINT := 45;  (* DEF[77].LWH[0]: Длина L *)
      MW777 AT %MW777 : UINT := 180;  (* DEF[77].LWH[1]: Ширина W *)
      MW778 AT %MW778 : UINT := 1700;  (* DEF[77].LWH[2]: Высота H *)
      MW779 AT %MW779 : UINT := 16#1100;  (* DEF[77].GMV: #Grd(4)|#Mat(4)|#Val(8) *)
      MW780 AT %MW780 : UINT := 16#4282;  (* DEF[78].ID: - Маслоканал-3 (прав) *)
      MW781 AT %MW781 : UINT := 16#400F;  (* DEF[78].CF: Флаги (СК|ось|форма) *)
      MW782 AT %MW782 : UINT := 0;  (* DEF[78].R0: Начальный радиус *)
      MW783 AT %MW783 : UINT := 545;  (* DEF[78].XYZ[0]: Координата X *)
      MW784 AT %MW784 : UINT := -90;  (* DEF[78].XYZ[1]: Координата Y *)
      MW785 AT %MW785 : UINT := 150;  (* DEF[78].XYZ[2]: Координата Z *)
      MW786 AT %MW786 : UINT := 45;  (* DEF[78].LWH[0]: Длина L *)
      MW787 AT %MW787 : UINT := 180;  (* DEF[78].LWH[1]: Ширина W *)
      MW788 AT %MW788 : UINT := 1700;  (* DEF[78].LWH[2]: Высота H *)
      MW789 AT %MW789 : UINT := 16#1100;  (* DEF[78].GMV: #Grd(4)|#Mat(4)|#Val(8) *)
      MW790 AT %MW790 : UINT := 16#4300;  (* DEF[79].ID: = Фаза 3 (прав) = *)
      MW791 AT %MW791 : UINT := 16#F006;  (* DEF[79].CF: Флаги (СК|ось|форма) *)
      MW792 AT %MW792 : UINT := 0;  (* DEF[79].R0: Начальный радиус *)
      MW793 AT %MW793 : UINT := 2950;  (* DEF[79].XYZ[0]: Координата X *)
      MW794 AT %MW794 : UINT := 590;  (* DEF[79].XYZ[1]: Координата Y *)
      MW795 AT %MW795 : UINT := 0;  (* DEF[79].XYZ[2]: Координата Z *)
      MW796 AT %MW796 : UINT := 590;  (* DEF[79].LWH[0]: Длина L *)
      MW797 AT %MW797 : UINT := 360;  (* DEF[79].LWH[1]: Ширина W *)
      MW798 AT %MW798 : UINT := 2000;  (* DEF[79].LWH[2]: Высота H *)
      MW799 AT %MW799 : UINT := 16#1000;  (* DEF[79].GMV: #Grd(4)|#Mat(4)|#Val(8) *)
      MW800 AT %MW800 : UINT := 16#4310;  (* DEF[80].ID: - Стержень *)
      MW801 AT %MW801 : UINT := 16#4000;  (* DEF[80].CF: Флаги (СК|ось|форма) *)
      MW802 AT %MW802 : UINT := 0;  (* DEF[80].R0: Начальный радиус *)
      MW803 AT %MW803 : UINT := 0;  (* DEF[80].XYZ[0]: Координата X *)
      MW804 AT %MW804 : UINT := 0;  (* DEF[80].XYZ[1]: Координата Y *)
      MW805 AT %MW805 : UINT := 0;  (* DEF[80].XYZ[2]: Координата Z *)
      MW806 AT %MW806 : UINT := 315;  (* DEF[80].LWH[0]: Длина L *)
      MW807 AT %MW807 : UINT := 360;  (* DEF[80].LWH[1]: Ширина W *)
      MW808 AT %MW808 : UINT := 2000;  (* DEF[80].LWH[2]: Высота H *)
      MW809 AT %MW809 : UINT := 16#1300;  (* DEF[80].GMV: #Grd(4)|#Mat(4)|#Val(8) *)
      MW810 AT %MW810 : UINT := 16#4320;  (* DEF[81].ID: - Масло сверху *)
      MW811 AT %MW811 : UINT := 16#4006;  (* DEF[81].CF: Флаги (СК|ось|форма) *)
      MW812 AT %MW812 : UINT := 0;  (* DEF[81].R0: Начальный радиус *)
      MW813 AT %MW813 : UINT := 315;  (* DEF[81].XYZ[0]: Координата X *)
      MW814 AT %MW814 : UINT := 0;  (* DEF[81].XYZ[1]: Координата Y *)
      MW815 AT %MW815 : UINT := 1850;  (* DEF[81].XYZ[2]: Координата Z *)
      MW816 AT %MW816 : UINT := 275;  (* DEF[81].LWH[0]: Длина L *)
      MW817 AT %MW817 : UINT := 360;  (* DEF[81].LWH[1]: Ширина W *)
      MW818 AT %MW818 : UINT := 150;  (* DEF[81].LWH[2]: Высота H *)
      MW819 AT %MW819 : UINT := 16#5100;  (* DEF[81].GMV: #Grd(4)|#Mat(4)|#Val(8) *)
      MW820 AT %MW820 : UINT := 16#4330;  (* DEF[82].ID: - Масло снизу *)
      MW821 AT %MW821 : UINT := 16#4006;  (* DEF[82].CF: Флаги (СК|ось|форма) *)
      MW822 AT %MW822 : UINT := 0;  (* DEF[82].R0: Начальный радиус *)
      MW823 AT %MW823 : UINT := 315;  (* DEF[82].XYZ[0]: Координата X *)
      MW824 AT %MW824 : UINT := 0;  (* DEF[82].XYZ[1]: Координата Y *)
      MW825 AT %MW825 : UINT := 0;  (* DEF[82].XYZ[2]: Координата Z *)
      MW826 AT %MW826 : UINT := 275;  (* DEF[82].LWH[0]: Длина L *)
      MW827 AT %MW827 : UINT := 360;  (* DEF[82].LWH[1]: Ширина W *)
      MW828 AT %MW828 : UINT := 150;  (* DEF[82].LWH[2]: Высота H *)
      MW829 AT %MW829 : UINT := 16#5100;  (* DEF[82].GMV: #Grd(4)|#Mat(4)|#Val(8) *)
      MW830 AT %MW830 : UINT := 16#4340;  (* DEF[83].ID: - Маслоканал-1 *)
      MW831 AT %MW831 : UINT := 16#4000;  (* DEF[83].CF: Флаги (СК|ось|форма) *)
      MW832 AT %MW832 : UINT := 0;  (* DEF[83].R0: Начальный радиус *)
      MW833 AT %MW833 : UINT := 315;  (* DEF[83].XYZ[0]: Координата X *)
      MW834 AT %MW834 : UINT := 0;  (* DEF[83].XYZ[1]: Координата Y *)
      MW835 AT %MW835 : UINT := 150;  (* DEF[83].XYZ[2]: Координата Z *)
      MW836 AT %MW836 : UINT := 30;  (* DEF[83].LWH[0]: Длина L *)
      MW837 AT %MW837 : UINT := 360;  (* DEF[83].LWH[1]: Ширина W *)
      MW838 AT %MW838 : UINT := 1700;  (* DEF[83].LWH[2]: Высота H *)
      MW839 AT %MW839 : UINT := 16#1100;  (* DEF[83].GMV: #Grd(4)|#Mat(4)|#Val(8) *)
      MW840 AT %MW840 : UINT := 16#4350;  (* DEF[84].ID: - Обмотка НН *)
      MW841 AT %MW841 : UINT := 16#4000;  (* DEF[84].CF: Флаги (СК|ось|форма) *)
      MW842 AT %MW842 : UINT := 0;  (* DEF[84].R0: Начальный радиус *)
      MW843 AT %MW843 : UINT := 345;  (* DEF[84].XYZ[0]: Координата X *)
      MW844 AT %MW844 : UINT := 0;  (* DEF[84].XYZ[1]: Координата Y *)
      MW845 AT %MW845 : UINT := 150;  (* DEF[84].XYZ[2]: Координата Z *)
      MW846 AT %MW846 : UINT := 80;  (* DEF[84].LWH[0]: Длина L *)
      MW847 AT %MW847 : UINT := 360;  (* DEF[84].LWH[1]: Ширина W *)
      MW848 AT %MW848 : UINT := 1700;  (* DEF[84].LWH[2]: Высота H *)
      MW849 AT %MW849 : UINT := 16#1400;  (* DEF[84].GMV: #Grd(4)|#Mat(4)|#Val(8) *)
      MW850 AT %MW850 : UINT := 16#4360;  (* DEF[85].ID: - Маслоканал-2 *)
      MW851 AT %MW851 : UINT := 16#4000;  (* DEF[85].CF: Флаги (СК|ось|форма) *)
      MW852 AT %MW852 : UINT := 0;  (* DEF[85].R0: Начальный радиус *)
      MW853 AT %MW853 : UINT := 425;  (* DEF[85].XYZ[0]: Координата X *)
      MW854 AT %MW854 : UINT := 0;  (* DEF[85].XYZ[1]: Координата Y *)
      MW855 AT %MW855 : UINT := 150;  (* DEF[85].XYZ[2]: Координата Z *)
      MW856 AT %MW856 : UINT := 30;  (* DEF[85].LWH[0]: Длина L *)
      MW857 AT %MW857 : UINT := 360;  (* DEF[85].LWH[1]: Ширина W *)
      MW858 AT %MW858 : UINT := 1700;  (* DEF[85].LWH[2]: Высота H *)
      MW859 AT %MW859 : UINT := 16#1100;  (* DEF[85].GMV: #Grd(4)|#Mat(4)|#Val(8) *)
      MW860 AT %MW860 : UINT := 16#4370;  (* DEF[86].ID: = Обмотка ВН = *)
      MW861 AT %MW861 : UINT := 16#C000;  (* DEF[86].CF: Флаги (СК|ось|форма) *)
      MW862 AT %MW862 : UINT := 0;  (* DEF[86].R0: Начальный радиус *)
      MW863 AT %MW863 : UINT := 455;  (* DEF[86].XYZ[0]: Координата X *)
      MW864 AT %MW864 : UINT := 0;  (* DEF[86].XYZ[1]: Координата Y *)
      MW865 AT %MW865 : UINT := 150;  (* DEF[86].XYZ[2]: Координата Z *)
      MW866 AT %MW866 : UINT := 90;  (* DEF[86].LWH[0]: Длина L *)
      MW867 AT %MW867 : UINT := 360;  (* DEF[86].LWH[1]: Ширина W *)
      MW868 AT %MW868 : UINT := 1700;  (* DEF[86].LWH[2]: Высота H *)
      MW869 AT %MW869 : UINT := 16#1000;  (* DEF[86].GMV: #Grd(4)|#Mat(4)|#Val(8) *)
      MW870 AT %MW870 : UINT := 16#4371;  (* DEF[87].ID: - Катушка ВН-1 *)
      MW871 AT %MW871 : UINT := 16#4000;  (* DEF[87].CF: Флаги (СК|ось|форма) *)
      MW872 AT %MW872 : UINT := 0;  (* DEF[87].R0: Начальный радиус *)
      MW873 AT %MW873 : UINT := 455;  (* DEF[87].XYZ[0]: Координата X *)
      MW874 AT %MW874 : UINT := 0;  (* DEF[87].XYZ[1]: Координата Y *)
      MW875 AT %MW875 : UINT := 150;  (* DEF[87].XYZ[2]: Координата Z *)
      MW876 AT %MW876 : UINT := 90;  (* DEF[87].LWH[0]: Длина L *)
      MW877 AT %MW877 : UINT := 360;  (* DEF[87].LWH[1]: Ширина W *)
      MW878 AT %MW878 : UINT := 170;  (* DEF[87].LWH[2]: Высота H *)
      MW879 AT %MW879 : UINT := 16#3500;  (* DEF[87].GMV: #Grd(4)|#Mat(4)|#Val(8) *)
      MW880 AT %MW880 : UINT := 16#4372;  (* DEF[88].ID: - Катушка ВН-2 *)
      MW881 AT %MW881 : UINT := 16#4000;  (* DEF[88].CF: Флаги (СК|ось|форма) *)
      MW882 AT %MW882 : UINT := 0;  (* DEF[88].R0: Начальный радиус *)
      MW883 AT %MW883 : UINT := 455;  (* DEF[88].XYZ[0]: Координата X *)
      MW884 AT %MW884 : UINT := 0;  (* DEF[88].XYZ[1]: Координата Y *)
      MW885 AT %MW885 : UINT := 320;  (* DEF[88].XYZ[2]: Координата Z *)
      MW886 AT %MW886 : UINT := 90;  (* DEF[88].LWH[0]: Длина L *)
      MW887 AT %MW887 : UINT := 360;  (* DEF[88].LWH[1]: Ширина W *)
      MW888 AT %MW888 : UINT := 170;  (* DEF[88].LWH[2]: Высота H *)
      MW889 AT %MW889 : UINT := 16#3500;  (* DEF[88].GMV: #Grd(4)|#Mat(4)|#Val(8) *)
      MW890 AT %MW890 : UINT := 16#4373;  (* DEF[89].ID: - Катушка ВН-3 *)
      MW891 AT %MW891 : UINT := 16#4000;  (* DEF[89].CF: Флаги (СК|ось|форма) *)
      MW892 AT %MW892 : UINT := 0;  (* DEF[89].R0: Начальный радиус *)
      MW893 AT %MW893 : UINT := 455;  (* DEF[89].XYZ[0]: Координата X *)
      MW894 AT %MW894 : UINT := 0;  (* DEF[89].XYZ[1]: Координата Y *)
      MW895 AT %MW895 : UINT := 490;  (* DEF[89].XYZ[2]: Координата Z *)
      MW896 AT %MW896 : UINT := 90;  (* DEF[89].LWH[0]: Длина L *)
      MW897 AT %MW897 : UINT := 360;  (* DEF[89].LWH[1]: Ширина W *)
      MW898 AT %MW898 : UINT := 170;  (* DEF[89].LWH[2]: Высота H *)
      MW899 AT %MW899 : UINT := 16#3500;  (* DEF[89].GMV: #Grd(4)|#Mat(4)|#Val(8) *)
      MW900 AT %MW900 : UINT := 16#4374;  (* DEF[90].ID: - Катушка ВН-4 *)
      MW901 AT %MW901 : UINT := 16#4000;  (* DEF[90].CF: Флаги (СК|ось|форма) *)
      MW902 AT %MW902 : UINT := 0;  (* DEF[90].R0: Начальный радиус *)
      MW903 AT %MW903 : UINT := 455;  (* DEF[90].XYZ[0]: Координата X *)
      MW904 AT %MW904 : UINT := 0;  (* DEF[90].XYZ[1]: Координата Y *)
      MW905 AT %MW905 : UINT := 660;  (* DEF[90].XYZ[2]: Координата Z *)
      MW906 AT %MW906 : UINT := 90;  (* DEF[90].LWH[0]: Длина L *)
      MW907 AT %MW907 : UINT := 360;  (* DEF[90].LWH[1]: Ширина W *)
      MW908 AT %MW908 : UINT := 170;  (* DEF[90].LWH[2]: Высота H *)
      MW909 AT %MW909 : UINT := 16#3500;  (* DEF[90].GMV: #Grd(4)|#Mat(4)|#Val(8) *)
      MW910 AT %MW910 : UINT := 16#4375;  (* DEF[91].ID: - Катушка ВН-5 *)
      MW911 AT %MW911 : UINT := 16#4000;  (* DEF[91].CF: Флаги (СК|ось|форма) *)
      MW912 AT %MW912 : UINT := 0;  (* DEF[91].R0: Начальный радиус *)
      MW913 AT %MW913 : UINT := 455;  (* DEF[91].XYZ[0]: Координата X *)
      MW914 AT %MW914 : UINT := 0;  (* DEF[91].XYZ[1]: Координата Y *)
      MW915 AT %MW915 : UINT := 830;  (* DEF[91].XYZ[2]: Координата Z *)
      MW916 AT %MW916 : UINT := 90;  (* DEF[91].LWH[0]: Длина L *)
      MW917 AT %MW917 : UINT := 360;  (* DEF[91].LWH[1]: Ширина W *)
      MW918 AT %MW918 : UINT := 170;  (* DEF[91].LWH[2]: Высота H *)
      MW919 AT %MW919 : UINT := 16#3500;  (* DEF[91].GMV: #Grd(4)|#Mat(4)|#Val(8) *)
      MW920 AT %MW920 : UINT := 16#4376;  (* DEF[92].ID: - Катушка ВН-6 *)
      MW921 AT %MW921 : UINT := 16#4000;  (* DEF[92].CF: Флаги (СК|ось|форма) *)
      MW922 AT %MW922 : UINT := 0;  (* DEF[92].R0: Начальный радиус *)
      MW923 AT %MW923 : UINT := 455;  (* DEF[92].XYZ[0]: Координата X *)
      MW924 AT %MW924 : UINT := 0;  (* DEF[92].XYZ[1]: Координата Y *)
      MW925 AT %MW925 : UINT := 1000;  (* DEF[92].XYZ[2]: Координата Z *)
      MW926 AT %MW926 : UINT := 90;  (* DEF[92].LWH[0]: Длина L *)
      MW927 AT %MW927 : UINT := 360;  (* DEF[92].LWH[1]: Ширина W *)
      MW928 AT %MW928 : UINT := 170;  (* DEF[92].LWH[2]: Высота H *)
      MW929 AT %MW929 : UINT := 16#3500;  (* DEF[92].GMV: #Grd(4)|#Mat(4)|#Val(8) *)
      MW930 AT %MW930 : UINT := 16#4377;  (* DEF[93].ID: - Катушка ВН-7 *)
      MW931 AT %MW931 : UINT := 16#4000;  (* DEF[93].CF: Флаги (СК|ось|форма) *)
      MW932 AT %MW932 : UINT := 0;  (* DEF[93].R0: Начальный радиус *)
      MW933 AT %MW933 : UINT := 455;  (* DEF[93].XYZ[0]: Координата X *)
      MW934 AT %MW934 : UINT := 0;  (* DEF[93].XYZ[1]: Координата Y *)
      MW935 AT %MW935 : UINT := 1170;  (* DEF[93].XYZ[2]: Координата Z *)
      MW936 AT %MW936 : UINT := 90;  (* DEF[93].LWH[0]: Длина L *)
      MW937 AT %MW937 : UINT := 360;  (* DEF[93].LWH[1]: Ширина W *)
      MW938 AT %MW938 : UINT := 170;  (* DEF[93].LWH[2]: Высота H *)
      MW939 AT %MW939 : UINT := 16#3500;  (* DEF[93].GMV: #Grd(4)|#Mat(4)|#Val(8) *)
      MW940 AT %MW940 : UINT := 16#4378;  (* DEF[94].ID: - Катушка ВН-8 *)
      MW941 AT %MW941 : UINT := 16#4000;  (* DEF[94].CF: Флаги (СК|ось|форма) *)
      MW942 AT %MW942 : UINT := 0;  (* DEF[94].R0: Начальный радиус *)
      MW943 AT %MW943 : UINT := 455;  (* DEF[94].XYZ[0]: Координата X *)
      MW944 AT %MW944 : UINT := 0;  (* DEF[94].XYZ[1]: Координата Y *)
      MW945 AT %MW945 : UINT := 1340;  (* DEF[94].XYZ[2]: Координата Z *)
      MW946 AT %MW946 : UINT := 90;  (* DEF[94].LWH[0]: Длина L *)
      MW947 AT %MW947 : UINT := 360;  (* DEF[94].LWH[1]: Ширина W *)
      MW948 AT %MW948 : UINT := 170;  (* DEF[94].LWH[2]: Высота H *)
      MW949 AT %MW949 : UINT := 16#3500;  (* DEF[94].GMV: #Grd(4)|#Mat(4)|#Val(8) *)
      MW950 AT %MW950 : UINT := 16#4379;  (* DEF[95].ID: - Катушка ВН-9 *)
      MW951 AT %MW951 : UINT := 16#4000;  (* DEF[95].CF: Флаги (СК|ось|форма) *)
      MW952 AT %MW952 : UINT := 0;  (* DEF[95].R0: Начальный радиус *)
      MW953 AT %MW953 : UINT := 455;  (* DEF[95].XYZ[0]: Координата X *)
      MW954 AT %MW954 : UINT := 0;  (* DEF[95].XYZ[1]: Координата Y *)
      MW955 AT %MW955 : UINT := 1510;  (* DEF[95].XYZ[2]: Координата Z *)
      MW956 AT %MW956 : UINT := 90;  (* DEF[95].LWH[0]: Длина L *)
      MW957 AT %MW957 : UINT := 360;  (* DEF[95].LWH[1]: Ширина W *)
      MW958 AT %MW958 : UINT := 170;  (* DEF[95].LWH[2]: Высота H *)
      MW959 AT %MW959 : UINT := 16#3500;  (* DEF[95].GMV: #Grd(4)|#Mat(4)|#Val(8) *)
      MW960 AT %MW960 : UINT := 16#437A;  (* DEF[96].ID: - Катушка ВН-10 *)
      MW961 AT %MW961 : UINT := 16#4000;  (* DEF[96].CF: Флаги (СК|ось|форма) *)
      MW962 AT %MW962 : UINT := 0;  (* DEF[96].R0: Начальный радиус *)
      MW963 AT %MW963 : UINT := 455;  (* DEF[96].XYZ[0]: Координата X *)
      MW964 AT %MW964 : UINT := 0;  (* DEF[96].XYZ[1]: Координата Y *)
      MW965 AT %MW965 : UINT := 1680;  (* DEF[96].XYZ[2]: Координата Z *)
      MW966 AT %MW966 : UINT := 90;  (* DEF[96].LWH[0]: Длина L *)
      MW967 AT %MW967 : UINT := 360;  (* DEF[96].LWH[1]: Ширина W *)
      MW968 AT %MW968 : UINT := 170;  (* DEF[96].LWH[2]: Высота H *)
      MW969 AT %MW969 : UINT := 16#3500;  (* DEF[96].GMV: #Grd(4)|#Mat(4)|#Val(8) *)
      MW970 AT %MW970 : UINT := 16#4380;  (* DEF[97].ID: = Маслоканал-3 = *)
      MW971 AT %MW971 : UINT := 16#C006;  (* DEF[97].CF: Флаги (СК|ось|форма) *)
      MW972 AT %MW972 : UINT := 0;  (* DEF[97].R0: Начальный радиус *)
      MW973 AT %MW973 : UINT := 545;  (* DEF[97].XYZ[0]: Координата X *)
      MW974 AT %MW974 : UINT := 0;  (* DEF[97].XYZ[1]: Координата Y *)
      MW975 AT %MW975 : UINT := 150;  (* DEF[97].XYZ[2]: Координата Z *)
      MW976 AT %MW976 : UINT := 45;  (* DEF[97].LWH[0]: Длина L *)
      MW977 AT %MW977 : UINT := 360;  (* DEF[97].LWH[1]: Ширина W *)
      MW978 AT %MW978 : UINT := 1700;  (* DEF[97].LWH[2]: Высота H *)
      MW979 AT %MW979 : UINT := 16#1000;  (* DEF[97].GMV: #Grd(4)|#Mat(4)|#Val(8) *)
      MW980 AT %MW980 : UINT := 16#4381;  (* DEF[98].ID: - Маслоканал-3 (лев) *)
      MW981 AT %MW981 : UINT := 16#4006;  (* DEF[98].CF: Флаги (СК|ось|форма) *)
      MW982 AT %MW982 : UINT := 0;  (* DEF[98].R0: Начальный радиус *)
      MW983 AT %MW983 : UINT := 545;  (* DEF[98].XYZ[0]: Координата X *)
      MW984 AT %MW984 : UINT := 90;  (* DEF[98].XYZ[1]: Координата Y *)
      MW985 AT %MW985 : UINT := 150;  (* DEF[98].XYZ[2]: Координата Z *)
      MW986 AT %MW986 : UINT := 45;  (* DEF[98].LWH[0]: Длина L *)
      MW987 AT %MW987 : UINT := 180;  (* DEF[98].LWH[1]: Ширина W *)
      MW988 AT %MW988 : UINT := 1700;  (* DEF[98].LWH[2]: Высота H *)
      MW989 AT %MW989 : UINT := 16#1100;  (* DEF[98].GMV: #Grd(4)|#Mat(4)|#Val(8) *)
      MW990 AT %MW990 : UINT := 16#4382;  (* DEF[99].ID: - Маслоканал-3 (прав) *)
      MW991 AT %MW991 : UINT := 16#4000;  (* DEF[99].CF: Флаги (СК|ось|форма) *)
      MW992 AT %MW992 : UINT := 0;  (* DEF[99].R0: Начальный радиус *)
      MW993 AT %MW993 : UINT := 545;  (* DEF[99].XYZ[0]: Координата X *)
      MW994 AT %MW994 : UINT := -90;  (* DEF[99].XYZ[1]: Координата Y *)
      MW995 AT %MW995 : UINT := 150;  (* DEF[99].XYZ[2]: Координата Z *)
      MW996 AT %MW996 : UINT := 45;  (* DEF[99].LWH[0]: Длина L *)
      MW997 AT %MW997 : UINT := 180;  (* DEF[99].LWH[1]: Ширина W *)
      MW998 AT %MW998 : UINT := 1700;  (* DEF[99].LWH[2]: Высота H *)
      MW999 AT %MW999 : UINT := 16#1100;  (* DEF[99].GMV: #Grd(4)|#Mat(4)|#Val(8) *)
      MW1000 AT %MW1000 : UINT := 0;  (* Резерв 0 *)
      MW1001 AT %MW1001 : UINT := 0;  (* Резерв 1 *)
      MW1002 AT %MW1002 : UINT := 0;  (* Резерв 2 *)
      MW1003 AT %MW1003 : UINT := 0;  (* Резерв 3 *)
      MW1004 AT %MW1004 : UINT := 0;  (* Резерв 4 *)
      MW1005 AT %MW1005 : UINT := 0;  (* Резерв 5 *)
      MW1006 AT %MW1006 : UINT := 0;  (* Резерв 6 *)
      MW1007 AT %MW1007 : UINT := 0;  (* Резерв 7 *)
      MW1008 AT %MW1008 : UINT := 0;  (* Резерв 8 *)
      MW1009 AT %MW1009 : UINT := 0;  (* Резерв 9 *)
      MW1010 AT %MW1010 : UINT := 0;  (* Резерв 10 *)
      MW1011 AT %MW1011 : UINT := 0;  (* Резерв 11 *)
      MW1012 AT %MW1012 : UINT := 0;  (* Резерв 12 *)
      MW1013 AT %MW1013 : UINT := 0;  (* Резерв 13 *)
      MW1014 AT %MW1014 : UINT := 0;  (* Резерв 14 *)
      MW1015 AT %MW1015 : UINT := 0;  (* Резерв 15 *)
      MW1016 AT %MW1016 : UINT := 0;  (* Резерв 16 *)
      MW1017 AT %MW1017 : UINT := 0;  (* Резерв 17 *)
      MW1018 AT %MW1018 : UINT := 0;  (* Резерв 18 *)
      MW1019 AT %MW1019 : UINT := 0;  (* Резерв 19 *)
      MW1020 AT %MW1020 : UINT := 0;  (* Резерв 20 *)
      MW1021 AT %MW1021 : UINT := 0;  (* Резерв 21 *)
      MW1022 AT %MW1022 : UINT := 0;  (* Резерв 22 *)
      MW1023 AT %MW1023 : UINT := 0;  (* Резерв 23 *)
      MD0 AT %MD0 : UDINT := 16#640A0600;  (* HEAD (Ni|Ng|Nm|Nv) *)
      MD1 AT %MD1 : UDINT := 16#01000000;  (* HEAD (Np|Ri|ID) *)
      MD2 AT %MD2 : UDINT := 16#00000000;  (* Заголовок. Слово 2 *)
      MD3 AT %MD3 : UDINT := 16#00000000;  (* Заголовок. Слово 3 *)
      MD4 AT %MD4 : UDINT := 16#00000000;  (* Заголовок. Слово 4 *)
      MD5 AT %MD5 : UDINT := 16#00000000;  (* Заголовок. Слово 5 *)
      MD6 AT %MD6 : UDINT := 16#00000000;  (* Заголовок. Слово 6 *)
      MD7 AT %MD7 : UDINT := 16#00000000;  (* Заголовок. Слово 7 *)
      MD8 AT %MD8 : UDINT := 16#00000000;  (* Заголовок. Слово 8 *)
      MD9 AT %MD9 : UDINT := 16#00000000;  (* Заголовок. Слово 9 *)
      MD10 AT %MD10 : UDINT := 16#08084000;  (* GRD[0] Сетка-0 *)
      MD11 AT %MD11 : UDINT := 16#08102000;  (* GRD[1] Сетка-1 *)
      MD12 AT %MD12 : UDINT := 16#08201000;  (* GRD[2] Сетка-2 *)
      MD13 AT %MD13 : UDINT := 16#08400800;  (* GRD[3] Сетка-3 *)
      MD14 AT %MD14 : UDINT := 16#10082000;  (* GRD[4] Сетка-4 *)
      MD15 AT %MD15 : UDINT := 16#10101000;  (* GRD[5] Сетка-5 *)
      MD16 AT %MD16 : UDINT := 16#10200800;  (* GRD[6] Сетка-6 *)
      MD17 AT %MD17 : UDINT := 16#20081000;  (* GRD[7] Сетка-7 *)
      MD18 AT %MD18 : UDINT := 16#20100800;  (* GRD[8] Сетка-8 *)
      MD19 AT %MD19 : UDINT := 16#40080800;  (* GRD[9] Сетка-9 *)
      MD20 AT %MD20 : UDINT := 16#FFFFFFFF;  (* GRD[10] Сетка-10 (Custom-0) *)
      MD21 AT %MD21 : UDINT := 16#FFFFFFFF;  (* GRD[11] Сетка-11 (Custom-1) *)
      MD22 AT %MD22 : UDINT := 1021719033;  (* MAT[0] К теплопроводности *)
      MD23 AT %MD23 : UDINT := 1148928000;  (* MAT[0] Уд. теплоемкость *)
      MD24 AT %MD24 : UDINT := 1067240653;  (* MAT[0] Плотность *)
      MD25 AT %MD25 : UDINT := 0;  (* MAT[0] Дин. вязкость *)
      MD26 AT %MD26 : UDINT := 1038254657;  (* MAT[1] К теплопроводности *)
      MD27 AT %MD27 : UDINT := 1154523136;  (* MAT[1] Уд. теплоемкость *)
      MD28 AT %MD28 : UDINT := 1146934067;  (* MAT[1] Плотность *)
      MD29 AT %MD29 : UDINT := 1017263004;  (* MAT[1] Дин. вязкость *)
      MD30 AT %MD30 : UDINT := 1112014848;  (* MAT[2] К теплопроводности *)
      MD31 AT %MD31 : UDINT := 1139146752;  (* MAT[2] Уд. теплоемкость *)
      MD32 AT %MD32 : UDINT := 1173536768;  (* MAT[2] Плотность *)
      MD33 AT %MD33 : UDINT := 0;  (* MAT[2] Дин. вязкость *)
      MD34 AT %MD34 : UDINT := 1110966272;  (* MAT[3] К теплопроводности *)
      MD35 AT %MD35 : UDINT := 1139802112;  (* MAT[3] Уд. теплоемкость *)
      MD36 AT %MD36 : UDINT := 1173295104;  (* MAT[3] Плотность *)
      MD37 AT %MD37 : UDINT := 0;  (* MAT[3] Дин. вязкость *)
      MD38 AT %MD38 : UDINT := 1137180672;  (* MAT[4] К теплопроводности *)
      MD39 AT %MD39 : UDINT := 1136689152;  (* MAT[4] Уд. теплоемкость *)
      MD40 AT %MD40 : UDINT := 1175163904;  (* MAT[4] Плотность *)
      MD41 AT %MD41 : UDINT := 0;  (* MAT[4] Дин. вязкость *)
      MD42 AT %MD42 : UDINT := 1137180672;  (* MAT[5] К теплопроводности *)
      MD43 AT %MD43 : UDINT := 1136689152;  (* MAT[5] Уд. теплоемкость *)
      MD44 AT %MD44 : UDINT := 1175163904;  (* MAT[5] Плотность *)
      MD45 AT %MD45 : UDINT := 0;  (* MAT[5] Дин. вязкость *)
      MD46 AT %MD46 : UDINT := 16#FFFFFFFF;  (* MAT[6] К теплопроводности *)
      MD47 AT %MD47 : UDINT := 16#FFFFFFFF;  (* MAT[6] Уд. теплоемкость *)
      MD48 AT %MD48 : UDINT := 16#FFFFFFFF;  (* MAT[6] Плотность *)
      MD49 AT %MD49 : UDINT := 16#FFFFFFFF;  (* MAT[6] Дин. вязкость *)
      MD50 AT %MD50 : UDINT := 16#FFFFFFFF;  (* MAT[7] К теплопроводности *)
      MD51 AT %MD51 : UDINT := 16#FFFFFFFF;  (* MAT[7] Уд. теплоемкость *)
      MD52 AT %MD52 : UDINT := 16#FFFFFFFF;  (* MAT[7] Плотность *)
      MD53 AT %MD53 : UDINT := 16#FFFFFFFF;  (* MAT[7] Дин. вязкость *)
      MD54 AT %MD54 : UDINT := 16#FFFFFFFF;  (* MAT[8] К теплопроводности *)
      MD55 AT %MD55 : UDINT := 16#FFFFFFFF;  (* MAT[8] Уд. теплоемкость *)
      MD56 AT %MD56 : UDINT := 16#FFFFFFFF;  (* MAT[8] Плотность *)
      MD57 AT %MD57 : UDINT := 16#FFFFFFFF;  (* MAT[8] Дин. вязкость *)
      MD58 AT %MD58 : UDINT := 16#FFFFFFFF;  (* MAT[9] К теплопроводности *)
      MD59 AT %MD59 : UDINT := 16#FFFFFFFF;  (* MAT[9] Уд. теплоемкость *)
      MD60 AT %MD60 : UDINT := 16#FFFFFFFF;  (* MAT[9] Плотность *)
      MD61 AT %MD61 : UDINT := 16#FFFFFFFF;  (* MAT[9] Дин. вязкость *)
      MD62 AT %MD62 : UDINT := 16#FFFFFFFF;  (* MAT[10] К теплопроводности *)
      MD63 AT %MD63 : UDINT := 16#FFFFFFFF;  (* MAT[10] Уд. теплоемкость *)
      MD64 AT %MD64 : UDINT := 16#FFFFFFFF;  (* MAT[10] Плотность *)
      MD65 AT %MD65 : UDINT := 16#FFFFFFFF;  (* MAT[10] Дин. вязкость *)
      MD66 AT %MD66 : UDINT := 16#FFFFFFFF;  (* MAT[11] К теплопроводности *)
      MD67 AT %MD67 : UDINT := 16#FFFFFFFF;  (* MAT[11] Уд. теплоемкость *)
      MD68 AT %MD68 : UDINT := 16#FFFFFFFF;  (* MAT[11] Плотность *)
      MD69 AT %MD69 : UDINT := 16#FFFFFFFF;  (* MAT[11] Дин. вязкость *)
      MD70 AT %MD70 : UDINT := 16#00000000;  (* VAL[0] Value-index | Part-Prof-X *)
      MD71 AT %MD71 : UDINT := 16#00000000;  (* VAL[0] Part-Prof-Y | Part-Prof-Z *)
      MD72 AT %MD72 : UDINT := 16#00000000;  (* VAL[1] Value-index | Part-Prof-X *)
      MD73 AT %MD73 : UDINT := 16#00000000;  (* VAL[1] Part-Prof-Y | Part-Prof-Z *)
      MD74 AT %MD74 : UDINT := 16#00000000;  (* VAL[2] Value-index | Part-Prof-X *)
      MD75 AT %MD75 : UDINT := 16#00000000;  (* VAL[2] Part-Prof-Y | Part-Prof-Z *)
      MD76 AT %MD76 : UDINT := 16#00000000;  (* VAL[3] Value-index | Part-Prof-X *)
      MD77 AT %MD77 : UDINT := 16#00000000;  (* VAL[3] Part-Prof-Y | Part-Prof-Z *)
      MD78 AT %MD78 : UDINT := 16#00000000;  (* VAL[4] Value-index | Part-Prof-X *)
      MD79 AT %MD79 : UDINT := 16#00000000;  (* VAL[4] Part-Prof-Y | Part-Prof-Z *)
      MD80 AT %MD80 : UDINT := 16#00000000;  (* VAL[5] Value-index | Part-Prof-X *)
      MD81 AT %MD81 : UDINT := 16#00000000;  (* VAL[5] Part-Prof-Y | Part-Prof-Z *)
      MD82 AT %MD82 : UDINT := 16#00000000;  (* VAL[6] Value-index | Part-Prof-X *)
      MD83 AT %MD83 : UDINT := 16#00000000;  (* VAL[6] Part-Prof-Y | Part-Prof-Z *)
      MD84 AT %MD84 : UDINT := 16#00000000;  (* VAL[7] Value-index | Part-Prof-X *)
      MD85 AT %MD85 : UDINT := 16#00000000;  (* VAL[7] Part-Prof-Y | Part-Prof-Z *)
      MD86 AT %MD86 : UDINT := 16#00000000;  (* VAL[8] Value-index | Part-Prof-X *)
      MD87 AT %MD87 : UDINT := 16#00000000;  (* VAL[8] Part-Prof-Y | Part-Prof-Z *)
      MD88 AT %MD88 : UDINT := 16#00000000;  (* VAL[9] Value-index | Part-Prof-X *)
      MD89 AT %MD89 : UDINT := 16#00000000;  (* VAL[9] Part-Prof-Y | Part-Prof-Z *)
      MD90 AT %MD90 : UDINT := 16#00000000;  (* VAL[10] Value-index | Part-Prof-X *)
      MD91 AT %MD91 : UDINT := 16#00000000;  (* VAL[10] Part-Prof-Y | Part-Prof-Z *)
      MD92 AT %MD92 : UDINT := 16#00000000;  (* VAL[11] Value-index | Part-Prof-X *)
      MD93 AT %MD93 : UDINT := 16#00000000;  (* VAL[11] Part-Prof-Y | Part-Prof-Z *)
      MD94 AT %MD94 : UDINT := 16#00000000;  (* VAL[12] Value-index | Part-Prof-X *)
      MD95 AT %MD95 : UDINT := 16#00000000;  (* VAL[12] Part-Prof-Y | Part-Prof-Z *)
      MD96 AT %MD96 : UDINT := 16#00000000;  (* VAL[13] Value-index | Part-Prof-X *)
      MD97 AT %MD97 : UDINT := 16#00000000;  (* VAL[13] Part-Prof-Y | Part-Prof-Z *)
      MD98 AT %MD98 : UDINT := 16#00000000;  (* VAL[14] Value-index | Part-Prof-X *)
      MD99 AT %MD99 : UDINT := 16#00000000;  (* VAL[14] Part-Prof-Y | Part-Prof-Z *)
      MD100 AT %MD100 : UDINT := 16#00000000;  (* VAL[15] Value-index | Part-Prof-X *)
      MD101 AT %MD101 : UDINT := 16#00000000;  (* VAL[15] Part-Prof-Y | Part-Prof-Z *)
      MD102 AT %MD102 : UDINT := 16#00000000;  (* VAL[16] Value-index | Part-Prof-X *)
      MD103 AT %MD103 : UDINT := 16#00000000;  (* VAL[16] Part-Prof-Y | Part-Prof-Z *)
      MD104 AT %MD104 : UDINT := 16#00000000;  (* VAL[17] Value-index | Part-Prof-X *)
      MD105 AT %MD105 : UDINT := 16#00000000;  (* VAL[17] Part-Prof-Y | Part-Prof-Z *)
      MD106 AT %MD106 : UDINT := 16#00000000;  (* VAL[18] Value-index | Part-Prof-X *)
      MD107 AT %MD107 : UDINT := 16#00000000;  (* VAL[18] Part-Prof-Y | Part-Prof-Z *)
      MD108 AT %MD108 : UDINT := 16#00000000;  (* VAL[19] Value-index | Part-Prof-X *)
      MD109 AT %MD109 : UDINT := 16#00000000;  (* VAL[19] Part-Prof-Y | Part-Prof-Z *)
      MD110 AT %MD110 : UDINT := 16#00000000;  (* VAL[20] Value-index | Part-Prof-X *)
      MD111 AT %MD111 : UDINT := 16#00000000;  (* VAL[20] Part-Prof-Y | Part-Prof-Z *)
      MD112 AT %MD112 : UDINT := 16#00000000;  (* VAL[21] Value-index | Part-Prof-X *)
      MD113 AT %MD113 : UDINT := 16#00000000;  (* VAL[21] Part-Prof-Y | Part-Prof-Z *)
      MD114 AT %MD114 : UDINT := 16#00000000;  (* VAL[22] Value-index | Part-Prof-X *)
      MD115 AT %MD115 : UDINT := 16#00000000;  (* VAL[22] Part-Prof-Y | Part-Prof-Z *)
      MD116 AT %MD116 : UDINT := 16#00000000;  (* VAL[23] Value-index | Part-Prof-X *)
      MD117 AT %MD117 : UDINT := 16#00000000;  (* VAL[23] Part-Prof-Y | Part-Prof-Z *)
      MD118 AT %MD118 : UDINT := 16#00000000;  (* VAL[24] Value-index | Part-Prof-X *)
      MD119 AT %MD119 : UDINT := 16#00000000;  (* VAL[24] Part-Prof-Y | Part-Prof-Z *)
      MD120 AT %MD120 : UDINT := 16#00000000;  (* PRO[0] A-B [0] | A-B [1] *)
      MD121 AT %MD121 : UDINT := 16#00000000;  (* PRO[0] A-B [2] | A-B [3] *)
      MD122 AT %MD122 : UDINT := 16#00000000;  (* PRO[0] A-B [4] | A-B [5] *)
      MD123 AT %MD123 : UDINT := 16#00000000;  (* PRO[0] A-B [6] | A-B [7] *)
      MD124 AT %MD124 : UDINT := 16#00000000;  (* PRO[0] A-B [8] | A-B [9] *)
      MD125 AT %MD125 : UDINT := 16#00000000;  (* PRO[0] A-B [10] | A-B [11] *)
      MD126 AT %MD126 : UDINT := 16#00000000;  (* PRO[1] A-B [0] | A-B [1] *)
      MD127 AT %MD127 : UDINT := 16#00000000;  (* PRO[1] A-B [2] | A-B [3] *)
      MD128 AT %MD128 : UDINT := 16#00000000;  (* PRO[1] A-B [4] | A-B [5] *)
      MD129 AT %MD129 : UDINT := 16#00000000;  (* PRO[1] A-B [6] | A-B [7] *)
      MD130 AT %MD130 : UDINT := 16#00000000;  (* PRO[1] A-B [8] | A-B [9] *)
      MD131 AT %MD131 : UDINT := 16#00000000;  (* PRO[1] A-B [10] | A-B [11] *)
      MD132 AT %MD132 : UDINT := 16#00000000;  (* PRO[2] A-B [0] | A-B [1] *)
      MD133 AT %MD133 : UDINT := 16#00000000;  (* PRO[2] A-B [2] | A-B [3] *)
      MD134 AT %MD134 : UDINT := 16#00000000;  (* PRO[2] A-B [4] | A-B [5] *)
      MD135 AT %MD135 : UDINT := 16#00000000;  (* PRO[2] A-B [6] | A-B [7] *)
      MD136 AT %MD136 : UDINT := 16#00000000;  (* PRO[2] A-B [8] | A-B [9] *)
      MD137 AT %MD137 : UDINT := 16#00000000;  (* PRO[2] A-B [10] | A-B [11] *)
      MD138 AT %MD138 : UDINT := 16#00000000;  (* PRO[3] A-B [0] | A-B [1] *)
      MD139 AT %MD139 : UDINT := 16#00000000;  (* PRO[3] A-B [2] | A-B [3] *)
      MD140 AT %MD140 : UDINT := 16#00000000;  (* PRO[3] A-B [4] | A-B [5] *)
      MD141 AT %MD141 : UDINT := 16#00000000;  (* PRO[3] A-B [6] | A-B [7] *)
      MD142 AT %MD142 : UDINT := 16#00000000;  (* PRO[3] A-B [8] | A-B [9] *)
      MD143 AT %MD143 : UDINT := 16#00000000;  (* PRO[3] A-B [10] | A-B [11] *)
      MD144 AT %MD144 : UDINT := 16#00000000;  (* PRO[4] A-B [0] | A-B [1] *)
      MD145 AT %MD145 : UDINT := 16#00000000;  (* PRO[4] A-B [2] | A-B [3] *)
      MD146 AT %MD146 : UDINT := 16#00000000;  (* PRO[4] A-B [4] | A-B [5] *)
      MD147 AT %MD147 : UDINT := 16#00000000;  (* PRO[4] A-B [6] | A-B [7] *)
      MD148 AT %MD148 : UDINT := 16#00000000;  (* PRO[4] A-B [8] | A-B [9] *)
      MD149 AT %MD149 : UDINT := 16#00000000;  (* PRO[4] A-B [10] | A-B [11] *)
      MD150 AT %MD150 : UDINT := 16#00000000;  (* PRO[5] A-B [0] | A-B [1] *)
      MD151 AT %MD151 : UDINT := 16#00000000;  (* PRO[5] A-B [2] | A-B [3] *)
      MD152 AT %MD152 : UDINT := 16#00000000;  (* PRO[5] A-B [4] | A-B [5] *)
      MD153 AT %MD153 : UDINT := 16#00000000;  (* PRO[5] A-B [6] | A-B [7] *)
      MD154 AT %MD154 : UDINT := 16#00000000;  (* PRO[5] A-B [8] | A-B [9] *)
      MD155 AT %MD155 : UDINT := 16#00000000;  (* PRO[5] A-B [10] | A-B [11] *)
      MD156 AT %MD156 : UDINT := 16#00000000;  (* PRO[6] A-B [0] | A-B [1] *)
      MD157 AT %MD157 : UDINT := 16#00000000;  (* PRO[6] A-B [2] | A-B [3] *)
      MD158 AT %MD158 : UDINT := 16#00000000;  (* PRO[6] A-B [4] | A-B [5] *)
      MD159 AT %MD159 : UDINT := 16#00000000;  (* PRO[6] A-B [6] | A-B [7] *)
      MD160 AT %MD160 : UDINT := 16#00000000;  (* PRO[6] A-B [8] | A-B [9] *)
      MD161 AT %MD161 : UDINT := 16#00000000;  (* PRO[6] A-B [10] | A-B [11] *)
      MD162 AT %MD162 : UDINT := 16#00000000;  (* PRO[7] A-B [0] | A-B [1] *)
      MD163 AT %MD163 : UDINT := 16#00000000;  (* PRO[7] A-B [2] | A-B [3] *)
      MD164 AT %MD164 : UDINT := 16#00000000;  (* PRO[7] A-B [4] | A-B [5] *)
      MD165 AT %MD165 : UDINT := 16#00000000;  (* PRO[7] A-B [6] | A-B [7] *)
      MD166 AT %MD166 : UDINT := 16#00000000;  (* PRO[7] A-B [8] | A-B [9] *)
      MD167 AT %MD167 : UDINT := 16#00000000;  (* PRO[7] A-B [10] | A-B [11] *)
      MD168 AT %MD168 : UDINT := 16#00000000;  (* PRO[8] A-B [0] | A-B [1] *)
      MD169 AT %MD169 : UDINT := 16#00000000;  (* PRO[8] A-B [2] | A-B [3] *)
      MD170 AT %MD170 : UDINT := 16#00000000;  (* PRO[8] A-B [4] | A-B [5] *)
      MD171 AT %MD171 : UDINT := 16#00000000;  (* PRO[8] A-B [6] | A-B [7] *)
      MD172 AT %MD172 : UDINT := 16#00000000;  (* PRO[8] A-B [8] | A-B [9] *)
      MD173 AT %MD173 : UDINT := 16#00000000;  (* PRO[8] A-B [10] | A-B [11] *)
      MD174 AT %MD174 : UDINT := 16#00000000;  (* PRO[9] A-B [0] | A-B [1] *)
      MD175 AT %MD175 : UDINT := 16#00000000;  (* PRO[9] A-B [2] | A-B [3] *)
      MD176 AT %MD176 : UDINT := 16#00000000;  (* PRO[9] A-B [4] | A-B [5] *)
      MD177 AT %MD177 : UDINT := 16#00000000;  (* PRO[9] A-B [6] | A-B [7] *)
      MD178 AT %MD178 : UDINT := 16#00000000;  (* PRO[9] A-B [8] | A-B [9] *)
      MD179 AT %MD179 : UDINT := 16#00000000;  (* PRO[9] A-B [10] | A-B [11] *)
      MD180 AT %MD180 : UDINT := 16#00000000;  (* PRO[10] A-B [0] | A-B [1] *)
      MD181 AT %MD181 : UDINT := 16#00000000;  (* PRO[10] A-B [2] | A-B [3] *)
      MD182 AT %MD182 : UDINT := 16#00000000;  (* PRO[10] A-B [4] | A-B [5] *)
      MD183 AT %MD183 : UDINT := 16#00000000;  (* PRO[10] A-B [6] | A-B [7] *)
      MD184 AT %MD184 : UDINT := 16#00000000;  (* PRO[10] A-B [8] | A-B [9] *)
      MD185 AT %MD185 : UDINT := 16#00000000;  (* PRO[10] A-B [10] | A-B [11] *)
      MD186 AT %MD186 : UDINT := 16#00000000;  (* PRO[11] A-B [0] | A-B [1] *)
      MD187 AT %MD187 : UDINT := 16#00000000;  (* PRO[11] A-B [2] | A-B [3] *)
      MD188 AT %MD188 : UDINT := 16#00000000;  (* PRO[11] A-B [4] | A-B [5] *)
      MD189 AT %MD189 : UDINT := 16#00000000;  (* PRO[11] A-B [6] | A-B [7] *)
      MD190 AT %MD190 : UDINT := 16#00000000;  (* PRO[11] A-B [8] | A-B [9] *)
      MD191 AT %MD191 : UDINT := 16#00000000;  (* PRO[11] A-B [10] | A-B [11] *)
      MD192 AT %MD192 : UDINT := 16#00000000;  (* PRO[12] A-B [0] | A-B [1] *)
      MD193 AT %MD193 : UDINT := 16#00000000;  (* PRO[12] A-B [2] | A-B [3] *)
      MD194 AT %MD194 : UDINT := 16#00000000;  (* PRO[12] A-B [4] | A-B [5] *)
      MD195 AT %MD195 : UDINT := 16#00000000;  (* PRO[12] A-B [6] | A-B [7] *)
      MD196 AT %MD196 : UDINT := 16#00000000;  (* PRO[12] A-B [8] | A-B [9] *)
      MD197 AT %MD197 : UDINT := 16#00000000;  (* PRO[12] A-B [10] | A-B [11] *)
      MD198 AT %MD198 : UDINT := 16#00000000;  (* PRO[13] A-B [0] | A-B [1] *)
      MD199 AT %MD199 : UDINT := 16#00000000;  (* PRO[13] A-B [2] | A-B [3] *)
      MD200 AT %MD200 : UDINT := 16#00000000;  (* PRO[13] A-B [4] | A-B [5] *)
      MD201 AT %MD201 : UDINT := 16#00000000;  (* PRO[13] A-B [6] | A-B [7] *)
      MD202 AT %MD202 : UDINT := 16#00000000;  (* PRO[13] A-B [8] | A-B [9] *)
      MD203 AT %MD203 : UDINT := 16#00000000;  (* PRO[13] A-B [10] | A-B [11] *)
      MD204 AT %MD204 : UDINT := 16#00000000;  (* PRO[14] A-B [0] | A-B [1] *)
      MD205 AT %MD205 : UDINT := 16#00000000;  (* PRO[14] A-B [2] | A-B [3] *)
      MD206 AT %MD206 : UDINT := 16#00000000;  (* PRO[14] A-B [4] | A-B [5] *)
      MD207 AT %MD207 : UDINT := 16#00000000;  (* PRO[14] A-B [6] | A-B [7] *)
      MD208 AT %MD208 : UDINT := 16#00000000;  (* PRO[14] A-B [8] | A-B [9] *)
      MD209 AT %MD209 : UDINT := 16#00000000;  (* PRO[14] A-B [10] | A-B [11] *)
      MD210 AT %MD210 : UDINT := 16#00000000;  (* PRO[15] A-B [0] | A-B [1] *)
      MD211 AT %MD211 : UDINT := 16#00000000;  (* PRO[15] A-B [2] | A-B [3] *)
      MD212 AT %MD212 : UDINT := 16#00000000;  (* PRO[15] A-B [4] | A-B [5] *)
      MD213 AT %MD213 : UDINT := 16#00000000;  (* PRO[15] A-B [6] | A-B [7] *)
      MD214 AT %MD214 : UDINT := 16#00000000;  (* PRO[15] A-B [8] | A-B [9] *)
      MD215 AT %MD215 : UDINT := 16#00000000;  (* PRO[15] A-B [10] | A-B [11] *)
      MD216 AT %MD216 : UDINT := 16#00000000;  (* PRO[16] A-B [0] | A-B [1] *)
      MD217 AT %MD217 : UDINT := 16#00000000;  (* PRO[16] A-B [2] | A-B [3] *)
      MD218 AT %MD218 : UDINT := 16#00000000;  (* PRO[16] A-B [4] | A-B [5] *)
      MD219 AT %MD219 : UDINT := 16#00000000;  (* PRO[16] A-B [6] | A-B [7] *)
      MD220 AT %MD220 : UDINT := 16#00000000;  (* PRO[16] A-B [8] | A-B [9] *)
      MD221 AT %MD221 : UDINT := 16#00000000;  (* PRO[16] A-B [10] | A-B [11] *)
      MD222 AT %MD222 : UDINT := 16#00000000;  (* PRO[17] A-B [0] | A-B [1] *)
      MD223 AT %MD223 : UDINT := 16#00000000;  (* PRO[17] A-B [2] | A-B [3] *)
      MD224 AT %MD224 : UDINT := 16#00000000;  (* PRO[17] A-B [4] | A-B [5] *)
      MD225 AT %MD225 : UDINT := 16#00000000;  (* PRO[17] A-B [6] | A-B [7] *)
      MD226 AT %MD226 : UDINT := 16#00000000;  (* PRO[17] A-B [8] | A-B [9] *)
      MD227 AT %MD227 : UDINT := 16#00000000;  (* PRO[17] A-B [10] | A-B [11] *)
      MD228 AT %MD228 : UDINT := 16#00000000;  (* PRO[18] A-B [0] | A-B [1] *)
      MD229 AT %MD229 : UDINT := 16#00000000;  (* PRO[18] A-B [2] | A-B [3] *)
      MD230 AT %MD230 : UDINT := 16#00000000;  (* PRO[18] A-B [4] | A-B [5] *)
      MD231 AT %MD231 : UDINT := 16#00000000;  (* PRO[18] A-B [6] | A-B [7] *)
      MD232 AT %MD232 : UDINT := 16#00000000;  (* PRO[18] A-B [8] | A-B [9] *)
      MD233 AT %MD233 : UDINT := 16#00000000;  (* PRO[18] A-B [10] | A-B [11] *)
      MD234 AT %MD234 : UDINT := 16#00000000;  (* PRO[19] A-B [0] | A-B [1] *)
      MD235 AT %MD235 : UDINT := 16#00000000;  (* PRO[19] A-B [2] | A-B [3] *)
      MD236 AT %MD236 : UDINT := 16#00000000;  (* PRO[19] A-B [4] | A-B [5] *)
      MD237 AT %MD237 : UDINT := 16#00000000;  (* PRO[19] A-B [6] | A-B [7] *)
      MD238 AT %MD238 : UDINT := 16#00000000;  (* PRO[19] A-B [8] | A-B [9] *)
      MD239 AT %MD239 : UDINT := 16#00000000;  (* PRO[19] A-B [10] | A-B [11] *)
      MD240 AT %MD240 : UDINT := 16#00000000;  (* PRO[20] A-B [0] | A-B [1] *)
      MD241 AT %MD241 : UDINT := 16#00000000;  (* PRO[20] A-B [2] | A-B [3] *)
      MD242 AT %MD242 : UDINT := 16#00000000;  (* PRO[20] A-B [4] | A-B [5] *)
      MD243 AT %MD243 : UDINT := 16#00000000;  (* PRO[20] A-B [6] | A-B [7] *)
      MD244 AT %MD244 : UDINT := 16#00000000;  (* PRO[20] A-B [8] | A-B [9] *)
      MD245 AT %MD245 : UDINT := 16#00000000;  (* PRO[20] A-B [10] | A-B [11] *)
      MD246 AT %MD246 : UDINT := 16#00000000;  (* PRO[21] A-B [0] | A-B [1] *)
      MD247 AT %MD247 : UDINT := 16#00000000;  (* PRO[21] A-B [2] | A-B [3] *)
      MD248 AT %MD248 : UDINT := 16#00000000;  (* PRO[21] A-B [4] | A-B [5] *)
      MD249 AT %MD249 : UDINT := 16#00000000;  (* PRO[21] A-B [6] | A-B [7] *)
      MD250 AT %MD250 : UDINT := 16#00000000;  (* PRO[21] A-B [8] | A-B [9] *)
      MD251 AT %MD251 : UDINT := 16#00000000;  (* PRO[21] A-B [10] | A-B [11] *)
      MD252 AT %MD252 : UDINT := 16#00000000;  (* PRO[22] A-B [0] | A-B [1] *)
      MD253 AT %MD253 : UDINT := 16#00000000;  (* PRO[22] A-B [2] | A-B [3] *)
      MD254 AT %MD254 : UDINT := 16#00000000;  (* PRO[22] A-B [4] | A-B [5] *)
      MD255 AT %MD255 : UDINT := 16#00000000;  (* PRO[22] A-B [6] | A-B [7] *)
      MD256 AT %MD256 : UDINT := 16#00000000;  (* PRO[22] A-B [8] | A-B [9] *)
      MD257 AT %MD257 : UDINT := 16#00000000;  (* PRO[22] A-B [10] | A-B [11] *)
      MD258 AT %MD258 : UDINT := 16#00000000;  (* PRO[23] A-B [0] | A-B [1] *)
      MD259 AT %MD259 : UDINT := 16#00000000;  (* PRO[23] A-B [2] | A-B [3] *)
      MD260 AT %MD260 : UDINT := 16#00000000;  (* PRO[23] A-B [4] | A-B [5] *)
      MD261 AT %MD261 : UDINT := 16#00000000;  (* PRO[23] A-B [6] | A-B [7] *)
      MD262 AT %MD262 : UDINT := 16#00000000;  (* PRO[23] A-B [8] | A-B [9] *)
      MD263 AT %MD263 : UDINT := 16#00000000;  (* PRO[23] A-B [10] | A-B [11] *)
      MD264 AT %MD264 : UDINT := 16#00000000;  (* PRO[24] A-B [0] | A-B [1] *)
      MD265 AT %MD265 : UDINT := 16#00000000;  (* PRO[24] A-B [2] | A-B [3] *)
      MD266 AT %MD266 : UDINT := 16#00000000;  (* PRO[24] A-B [4] | A-B [5] *)
      MD267 AT %MD267 : UDINT := 16#00000000;  (* PRO[24] A-B [6] | A-B [7] *)
      MD268 AT %MD268 : UDINT := 16#00000000;  (* PRO[24] A-B [8] | A-B [9] *)
      MD269 AT %MD269 : UDINT := 16#00000000;  (* PRO[24] A-B [10] | A-B [11] *)
      MD270 AT %MD270 : UDINT := 16#00000000;  (* PRO[25] A-B [0] | A-B [1] *)
      MD271 AT %MD271 : UDINT := 16#00000000;  (* PRO[25] A-B [2] | A-B [3] *)
      MD272 AT %MD272 : UDINT := 16#00000000;  (* PRO[25] A-B [4] | A-B [5] *)
      MD273 AT %MD273 : UDINT := 16#00000000;  (* PRO[25] A-B [6] | A-B [7] *)
      MD274 AT %MD274 : UDINT := 16#00000000;  (* PRO[25] A-B [8] | A-B [9] *)
      MD275 AT %MD275 : UDINT := 16#00000000;  (* PRO[25] A-B [10] | A-B [11] *)
      MD276 AT %MD276 : UDINT := 16#00000000;  (* PRO[26] A-B [0] | A-B [1] *)
      MD277 AT %MD277 : UDINT := 16#00000000;  (* PRO[26] A-B [2] | A-B [3] *)
      MD278 AT %MD278 : UDINT := 16#00000000;  (* PRO[26] A-B [4] | A-B [5] *)
      MD279 AT %MD279 : UDINT := 16#00000000;  (* PRO[26] A-B [6] | A-B [7] *)
      MD280 AT %MD280 : UDINT := 16#00000000;  (* PRO[26] A-B [8] | A-B [9] *)
      MD281 AT %MD281 : UDINT := 16#00000000;  (* PRO[26] A-B [10] | A-B [11] *)
      MD282 AT %MD282 : UDINT := 16#00000000;  (* PRO[27] A-B [0] | A-B [1] *)
      MD283 AT %MD283 : UDINT := 16#00000000;  (* PRO[27] A-B [2] | A-B [3] *)
      MD284 AT %MD284 : UDINT := 16#00000000;  (* PRO[27] A-B [4] | A-B [5] *)
      MD285 AT %MD285 : UDINT := 16#00000000;  (* PRO[27] A-B [6] | A-B [7] *)
      MD286 AT %MD286 : UDINT := 16#00000000;  (* PRO[27] A-B [8] | A-B [9] *)
      MD287 AT %MD287 : UDINT := 16#00000000;  (* PRO[27] A-B [10] | A-B [11] *)
      MD288 AT %MD288 : UDINT := 16#00000000;  (* PRO[28] A-B [0] | A-B [1] *)
      MD289 AT %MD289 : UDINT := 16#00000000;  (* PRO[28] A-B [2] | A-B [3] *)
      MD290 AT %MD290 : UDINT := 16#00000000;  (* PRO[28] A-B [4] | A-B [5] *)
      MD291 AT %MD291 : UDINT := 16#00000000;  (* PRO[28] A-B [6] | A-B [7] *)
      MD292 AT %MD292 : UDINT := 16#00000000;  (* PRO[28] A-B [8] | A-B [9] *)
      MD293 AT %MD293 : UDINT := 16#00000000;  (* PRO[28] A-B [10] | A-B [11] *)
      MD294 AT %MD294 : UDINT := 16#00000000;  (* PRO[29] A-B [0] | A-B [1] *)
      MD295 AT %MD295 : UDINT := 16#00000000;  (* PRO[29] A-B [2] | A-B [3] *)
      MD296 AT %MD296 : UDINT := 16#00000000;  (* PRO[29] A-B [4] | A-B [5] *)
      MD297 AT %MD297 : UDINT := 16#00000000;  (* PRO[29] A-B [6] | A-B [7] *)
      MD298 AT %MD298 : UDINT := 16#00000000;  (* PRO[29] A-B [8] | A-B [9] *)
      MD299 AT %MD299 : UDINT := 16#00000000;  (* PRO[29] A-B [10] | A-B [11] *)
      MD300 AT %MD300 : UDINT := 16#00000000;  (* CFG.Ns: N стерж.| CFG.Nr: N тип.рад *)
      MD301 AT %MD301 : UDINT := 16#00000000;  (* CFG.Tc: Период расчёта *)
      MD302 AT %MD302 : UDINT := 16#00000000;  (* RAD[0].Vm: Объем радиатора *)
      MD303 AT %MD303 : UDINT := 16#00000000;  (* RAD[0].Fk: Площадь конвекции *)
      MD304 AT %MD304 : UDINT := 16#00000000;  (* RAD[0].Q0: Расход своб конвекции *)
      MD305 AT %MD305 : UDINT := 16#00000000;  (* RAD[0].Q1: Расход принуд конвекции *)
      MD306 AT %MD306 : UDINT := 16#00000000;  (* RAD[0].Bl[0]: Vобдува- 1 вентилятор *)
      MD307 AT %MD307 : UDINT := 16#00000000;  (* RAD[0].Bl[1]: Vобдува- 2 вентилятора *)
      MD308 AT %MD308 : UDINT := 16#00000000;  (* RAD[0].Bl[2]: Vобдува- 3 вентилятора *)
      MD309 AT %MD309 : UDINT := 16#00000000;  (* RAD[0].Bl[3]: Vобдува- 4 вентилятора *)
      MD310 AT %MD310 : UDINT := 16#00000000;  (* RAD[1].Vm: Объем радиатора *)
